LIN {X 0,Y 412.608,Z 386.941,A -85,B 0,C 180,E1 -10561.189,E2 -10561.189} C_VEL
LIN {X 0,Y 413.421,Z 375.355,A -85,B 0,C 180,E1 -10564.715,E2 -10564.715} C_VEL
LIN {X 0,Y 413.845,Z 369.744,A -85,B 0,C 180,E1 -10566.469,E2 -10566.469} C_VEL
LIN {X 0,Y 413.178,Z 364.821,A -85,B 0,C 180,E1 -10568.11,E2 -10568.11} C_VEL
LIN {X 0,Y 411.531,Z 355.758,A -85,B 0,C 180,E1 -10571.286,E2 -10571.286} C_VEL
LIN {X 0,Y 411.225,Z 354.264,A -85,B 0,C 180,E1 -10571.883,E2 -10571.883} C_VEL
LIN {X 0,Y 411.182,Z 354.268,A -85,B 0,C 180,E1 -10575.51,E2 -10575.51} C_VEL
LIN {X 0,Y 411.168,Z 354.271,A -85,B 0,C 180,E1 -10578.772,E2 -10578.772} C_VEL
LIN {X 0,Y 411.21,Z 354.262,A -85,B 0,C 180,E1 -10581.832,E2 -10581.832} C_VEL
LIN {X 0,Y 411.215,Z 354.264,A -85,B 0,C 180,E1 -10585.122,E2 -10585.122} C_VEL
LIN {X 0,Y 411.171,Z 354.266,A -85,B 0,C 180,E1 -10588.003,E2 -10588.003} C_VEL
LIN {X 0,Y 411.223,Z 354.261,A -85,B 0,C 180,E1 -10591.41,E2 -10591.41} C_VEL
LIN {X 0,Y 411.243,Z 354.257,A -85,B 0,C 180,E1 -10593.62,E2 -10593.62} C_VEL
LIN {X 0,Y 411.209,Z 354.265,A -85,B 0,C 180,E1 -10596.853,E2 -10596.853} C_VEL
LIN {X 0,Y 411.22,Z 354.262,A -85,B 0,C 180,E1 -10600.051,E2 -10600.051} C_VEL
LIN {X 0,Y 411.268,Z 354.255,A -85,B 0,C 180,E1 -10603.132,E2 -10603.132} C_VEL
LIN {X 0,Y 411.311,Z 354.252,A -85,B 0,C 180,E1 -10606.896,E2 -10606.896} C_VEL
LIN {X 0,Y 411.298,Z 354.254,A -85,B 0,C 180,E1 -10610.162,E2 -10610.162} C_VEL
LIN {X 0,Y 411.488,Z 354.23,A -85,B 0,C 180,E1 -10612.147,E2 -10612.147} C_VEL
LIN {X 0,Y 411.481,Z 354.231,A -85,B 0,C 180,E1 -10614.118,E2 -10614.118} C_VEL
LIN {X 0,Y 411.517,Z 354.227,A -85,B 0,C 180,E1 -10618.043,E2 -10618.043} C_VEL
LIN {X 0,Y 411.648,Z 354.21,A -85,B 0,C 180,E1 -10620,E2 -10620} C_VEL
LIN {X 0,Y 411.463,Z 354.23,A -85,B 0,C 180,E1 -10622.937,E2 -10622.937} C_VEL
LIN {X 0,Y 411.467,Z 354.229,A -85,B 0,C 180,E1 -10626.867,E2 -10626.867} C_VEL
LIN {X 0,Y 411.3,Z 354.254,A -85,B 0,C 180,E1 -10629.839,E2 -10629.839} C_VEL
LIN {X 0,Y 411.312,Z 354.249,A -85,B 0,C 180,E1 -10633.104,E2 -10633.104} C_VEL
LIN {X 0,Y 411.264,Z 354.255,A -85,B 0,C 180,E1 -10636.889,E2 -10636.889} C_VEL
LIN {X 0,Y 411.237,Z 354.262,A -85,B 0,C 180,E1 -10639.987,E2 -10639.987} C_VEL
LIN {X 0,Y 411.21,Z 354.262,A -85,B 0,C 180,E1 -10643.148,E2 -10643.148} C_VEL
LIN {X 0,Y 411.244,Z 354.258,A -85,B 0,C 180,E1 -10646.381,E2 -10646.381} C_VEL
LIN {X 0,Y 411.207,Z 354.266,A -85,B 0,C 180,E1 -10649.713,E2 -10649.713} C_VEL
LIN {X 0,Y 411.213,Z 354.264,A -85,B 0,C 180,E1 -10653.156,E2 -10653.156} C_VEL
LIN {X 0,Y 411.199,Z 354.263,A -85,B 0,C 180,E1 -10656.553,E2 -10656.553} C_VEL
LIN {X 0,Y 411.221,Z 354.264,A -85,B 0,C 180,E1 -10659.728,E2 -10659.728} C_VEL
LIN {X 0,Y 411.18,Z 354.269,A -85,B 0,C 180,E1 -10663.133,E2 -10663.133} C_VEL
LIN {X 0,Y 411.174,Z 354.267,A -85,B 0,C 180,E1 -10665.881,E2 -10665.881} C_VEL
LIN {X 0,Y 411.17,Z 354.268,A -85,B 0,C 180,E1 -10668.771,E2 -10668.771} C_VEL
LIN {X 0,Y 411.21,Z 354.262,A -85,B 0,C 180,E1 -10671.831,E2 -10671.831} C_VEL
LIN {X 0,Y 411.217,Z 354.265,A -85,B 0,C 180,E1 -10675.121,E2 -10675.121} C_VEL
LIN {X 0,Y 411.172,Z 354.266,A -85,B 0,C 180,E1 -10678.002,E2 -10678.002} C_VEL
LIN {X 0,Y 411.225,Z 354.262,A -85,B 0,C 180,E1 -10681.41,E2 -10681.41} C_VEL
LIN {X 0,Y 411.244,Z 354.258,A -85,B 0,C 180,E1 -10683.619,E2 -10683.619} C_VEL
LIN {X 0,Y 411.21,Z 354.265,A -85,B 0,C 180,E1 -10686.852,E2 -10686.852} C_VEL
LIN {X 0,Y 411.221,Z 354.26,A -85,B 0,C 180,E1 -10690.05,E2 -10690.05} C_VEL
LIN {X 0,Y 411.269,Z 354.257,A -85,B 0,C 180,E1 -10693.131,E2 -10693.131} C_VEL
LIN {X 0,Y 411.312,Z 354.253,A -85,B 0,C 180,E1 -10696.895,E2 -10696.895} C_VEL
LIN {X 0,Y 411.3,Z 354.253,A -85,B 0,C 180,E1 -10700.161,E2 -10700.161} C_VEL
LIN {X 0,Y 411.393,Z 354.352,A -85,B 0,C 180,E1 -10701.301,E2 -10701.301} C_VEL
LIN {X 0,Y 414.802,Z 366.071,A -85,B 0,C 180,E1 -10702.018,E2 -10702.018} C_VEL
LIN {X 0,Y 415.459,Z 369.039,A -85,B 0,C 180,E1 -10702.222,E2 -10702.222} C_VEL
LIN {X 0,Y 414.97,Z 381.177,A -85,B 0,C 180,E1 -10703.069,E2 -10703.069} C_VEL
LIN {X 0,Y 414.349,Z 392.048,A -85,B 0,C 180,E1 -10704.036,E2 -10704.036} C_VEL
LIN {X 0,Y 413.737,Z 401.829,A -85,B 0,C 180,E1 -10705.127,E2 -10705.127} C_VEL
LIN {X 0,Y 413.111,Z 410.706,A -85,B 0,C 180,E1 -10706.342,E2 -10706.342} C_VEL
LIN {X 0,Y 412.467,Z 419.368,A -85,B 0,C 180,E1 -10707.802,E2 -10707.802} C_VEL
LIN {X 0,Y 411.878,Z 426.341,A -85,B 0,C 180,E1 -10709.266,E2 -10709.266} C_VEL
LIN {X 0,Y 411.557,Z 431.041,A -85,B 0,C 180,E1 -10710.489,E2 -10710.489} C_VEL
LIN {X 0,Y 411.291,Z 435.602,A -85,B 0,C 180,E1 -10711.958,E2 -10711.958} C_VEL
LIN {X 0,Y 411.045,Z 438.063,A -85,B 0,C 180,E1 -10712.939,E2 -10712.939} C_VEL
LIN {X 0,Y 410.904,Z 440.046,A -85,B 0,C 180,E1 -10713.922,E2 -10713.922} C_VEL
LIN {X 0,Y 410.94,Z 441.605,A -85,B 0,C 180,E1 -10714.905,E2 -10714.905} C_VEL
LIN {X 0,Y 410.84,Z 443.383,A -85,B 0,C 180,E1 -10716.667,E2 -10716.667} C_VEL
LIN {X 0,Y 410.829,Z 443.911,A -85,B 0,C 180,E1 -10717.865,E2 -10717.865} C_VEL
LIN {X 0,Y 410.835,Z 443.521,A -85,B 0,C 180,E1 -10719.849,E2 -10719.849} C_VEL
LIN {X 0,Y 410.913,Z 442.591,A -85,B 0,C 180,E1 -10720.928,E2 -10720.928} C_VEL
LIN {X 0,Y 410.347,Z 441.725,A -85,B 0,C 180,E1 -10721.738,E2 -10721.738} C_VEL
LIN {X 0,Y 407.723,Z 439.991,A -85,B 0,C 180,E1 -10723.059,E2 -10723.059} C_VEL
LIN {X 0,Y 405.184,Z 437.619,A -85,B 0,C 180,E1 -10724.37,E2 -10724.37} C_VEL
LIN {X 0,Y 404.754,Z 435.61,A -85,B 0,C 180,E1 -10725.154,E2 -10725.154} C_VEL
LIN {X 0,Y 405.227,Z 430.899,A -85,B 0,C 180,E1 -10726.628,E2 -10726.628} C_VEL
LIN {X 0,Y 405.873,Z 424.706,A -85,B 0,C 180,E1 -10728.16,E2 -10728.16} C_VEL
LIN {X 0,Y 406.622,Z 416.874,A -85,B 0,C 180,E1 -10729.696,E2 -10729.696} C_VEL
LIN {X 0,Y 407.382,Z 408.814,A -85,B 0,C 180,E1 -10730.975,E2 -10730.975} C_VEL
LIN {X 0,Y 408.129,Z 398.91,A -85,B 0,C 180,E1 -10732.261,E2 -10732.261} C_VEL
LIN {X 0,Y 408.883,Z 389.085,A -85,B 0,C 180,E1 -10733.286,E2 -10733.286} C_VEL
LIN {X 0,Y 409.693,Z 378.177,A -85,B 0,C 180,E1 -10734.187,E2 -10734.187} C_VEL
LIN {X 0,Y 409.807,Z 371.736,A -85,B 0,C 180,E1 -10734.641,E2 -10734.641} C_VEL
LIN {X 0,Y 405.955,Z 360.3,A -85,B 0,C 180,E1 -10735.523,E2 -10735.523} C_VEL
LIN {X 0,Y 404.213,Z 355.137,A -85,B 0,C 180,E1 -10735.867,E2 -10735.867} C_VEL
LIN {X 0,Y 404.178,Z 355.143,A -85,B 0,C 180,E1 -10739.135,E2 -10739.135} C_VEL
LIN {X 0,Y 404.142,Z 355.149,A -85,B 0,C 180,E1 -10742.621,E2 -10742.621} C_VEL
LIN {X 0,Y 404.181,Z 355.143,A -85,B 0,C 180,E1 -10745.189,E2 -10745.189} C_VEL
LIN {X 0,Y 404.156,Z 355.145,A -85,B 0,C 180,E1 -10748.756,E2 -10748.756} C_VEL
LIN {X 0,Y 404.124,Z 355.146,A -85,B 0,C 180,E1 -10751.599,E2 -10751.599} C_VEL
LIN {X 0,Y 404.148,Z 355.144,A -85,B 0,C 180,E1 -10754.522,E2 -10754.522} C_VEL
LIN {X 0,Y 404.17,Z 355.14,A -85,B 0,C 180,E1 -10757.299,E2 -10757.299} C_VEL
LIN {X 0,Y 404.167,Z 355.141,A -85,B 0,C 180,E1 -10759.955,E2 -10759.955} C_VEL
LIN {X 0,Y 404.14,Z 355.145,A -85,B 0,C 180,E1 -10763.123,E2 -10763.123} C_VEL
LIN {X 0,Y 404.143,Z 355.145,A -85,B 0,C 180,E1 -10766.187,E2 -10766.187} C_VEL
LIN {X 0,Y 404.153,Z 355.118,A -85,B 0,C 180,E1 -10769.715,E2 -10769.715} C_VEL
LIN {X 0,Y 404.193,Z 355.135,A -85,B 0,C 180,E1 -10773.122,E2 -10773.122} C_VEL
LIN {X 0,Y 404.175,Z 355.139,A -85,B 0,C 180,E1 -10775.334,E2 -10775.334} C_VEL
LIN {X 0,Y 404.136,Z 355.145,A -85,B 0,C 180,E1 -10778.58,E2 -10778.58} C_VEL
LIN {X 0,Y 404.207,Z 355.13,A -85,B 0,C 180,E1 -10781.761,E2 -10781.761} C_VEL
LIN {X 0,Y 404.205,Z 355.137,A -85,B 0,C 180,E1 -10784.882,E2 -10784.882} C_VEL
LIN {X 0,Y 404.268,Z 355.129,A -85,B 0,C 180,E1 -10787.959,E2 -10787.959} C_VEL
LIN {X 0,Y 404.43,Z 355.109,A -85,B 0,C 180,E1 -10792.099,E2 -10792.099} C_VEL
LIN {X 0,Y 404.421,Z 355.102,A -85,B 0,C 180,E1 -10794.015,E2 -10794.015} C_VEL
LIN {X 0,Y 404.48,Z 355.102,A -85,B 0,C 180,E1 -10798.008,E2 -10798.008} C_VEL
LIN {X 0,Y 404.61,Z 355.079,A -85,B 0,C 180,E1 -10800,E2 -10800} C_VEL
LIN {X 0,Y 404.42,Z 355.111,A -85,B 0,C 180,E1 -10802.988,E2 -10802.988} C_VEL
LIN {X 0,Y 404.408,Z 355.111,A -85,B 0,C 180,E1 -10806.987,E2 -10806.987} C_VEL
LIN {X 0,Y 404.255,Z 355.124,A -85,B 0,C 180,E1 -10810.012,E2 -10810.012} C_VEL
LIN {X 0,Y 404.262,Z 355.127,A -85,B 0,C 180,E1 -10813.211,E2 -10813.211} C_VEL
LIN {X 0,Y 404.211,Z 355.135,A -85,B 0,C 180,E1 -10817.007,E2 -10817.007} C_VEL
LIN {X 0,Y 404.16,Z 355.141,A -85,B 0,C 180,E1 -10820.352,E2 -10820.352} C_VEL
LIN {X 0,Y 404.166,Z 355.14,A -85,B 0,C 180,E1 -10823.575,E2 -10823.575} C_VEL
LIN {X 0,Y 404.18,Z 355.142,A -85,B 0,C 180,E1 -10825.767,E2 -10825.767} C_VEL
LIN {X 0,Y 404.194,Z 355.142,A -85,B 0,C 180,E1 -10828,E2 -10828} C_VEL
LIN {X 0,Y 404.14,Z 355.147,A -85,B 0,C 180,E1 -10831.559,E2 -10831.559} C_VEL
LIN {X 0,Y 404.182,Z 355.141,A -85,B 0,C 180,E1 -10835.016,E2 -10835.016} C_VEL
LIN {X 0,Y 404.161,Z 355.134,A -85,B 0,C 180,E1 -10838.756,E2 -10838.756} C_VEL
LIN {X 0,Y 404.188,Z 355.131,A -85,B 0,C 180,E1 -10841.611,E2 -10841.611} C_VEL
LIN {X 0,Y 404.196,Z 355.133,A -85,B 0,C 180,E1 -10844.53,E2 -10844.53} C_VEL
LIN {X 0,Y 404.204,Z 355.236,A -85,B 0,C 180,E1 -10846.112,E2 -10846.112} C_VEL
LIN {X 0,Y 405.964,Z 363.942,A -85,B 0,C 180,E1 -10849.616,E2 -10849.616} C_VEL
LIN {X 0,Y 407.483,Z 372.651,A -85,B 0,C 180,E1 -10852.869,E2 -10852.869} C_VEL
LIN {X 0,Y 407.297,Z 376.542,A -85,B 0,C 180,E1 -10854.193,E2 -10854.193} C_VEL
LIN {X 0,Y 406.171,Z 388.134,A -85,B 0,C 180,E1 -10857.979,E2 -10857.979} C_VEL
LIN {X 0,Y 405.429,Z 397.585,A -85,B 0,C 180,E1 -10860.964,E2 -10860.964} C_VEL
LIN {X 0,Y 404.756,Z 408.327,A -85,B 0,C 180,E1 -10864.274,E2 -10864.274} C_VEL
LIN {X 0,Y 404.112,Z 420.824,A -85,B 0,C 180,E1 -10868.044,E2 -10868.044} C_VEL
LIN {X 0,Y 403.632,Z 433.192,A -85,B 0,C 180,E1 -10871.703,E2 -10871.703} C_VEL
LIN {X 0,Y 405.744,Z 447.481,A -85,B 0,C 180,E1 -10872.223,E2 -10872.223} C_VEL
LIN {X 0,Y 406.862,Z 460.005,A -85,B 0,C 180,E1 -10872.843,E2 -10872.843} C_VEL
LIN {X 0,Y 407.384,Z 471.723,A -85,B 0,C 180,E1 -10873.592,E2 -10873.592} C_VEL
LIN {X 0,Y 406.784,Z 481.584,A -85,B 0,C 180,E1 -10874.339,E2 -10874.339} C_VEL
LIN {X 0,Y 405.845,Z 492.192,A -85,B 0,C 180,E1 -10875.33,E2 -10875.33} C_VEL
LIN {X 0,Y 405.155,Z 501.778,A -85,B 0,C 180,E1 -10876.435,E2 -10876.435} C_VEL
LIN {X 0,Y 404.349,Z 510.869,A -85,B 0,C 180,E1 -10877.707,E2 -10877.707} C_VEL
LIN {X 0,Y 403.745,Z 519.623,A -85,B 0,C 180,E1 -10879.216,E2 -10879.216} C_VEL
LIN {X 0,Y 403.409,Z 526.669,A -85,B 0,C 180,E1 -10880.727,E2 -10880.727} C_VEL
LIN {X 0,Y 403.217,Z 533.185,A -85,B 0,C 180,E1 -10882.489,E2 -10882.489} C_VEL
LIN {X 0,Y 403.256,Z 537.494,A -85,B 0,C 180,E1 -10883.998,E2 -10883.998} C_VEL
LIN {X 0,Y 403.23,Z 539.778,A -85,B 0,C 180,E1 -10885.001,E2 -10885.001} C_VEL
LIN {X 0,Y 403.368,Z 541.589,A -85,B 0,C 180,E1 -10886.004,E2 -10886.004} C_VEL
LIN {X 0,Y 403.421,Z 542.973,A -85,B 0,C 180,E1 -10887.005,E2 -10887.005} C_VEL
LIN {X 0,Y 403.367,Z 543.94,A -85,B 0,C 180,E1 -10888.004,E2 -10888.004} C_VEL
LIN {X 0,Y 403.382,Z 544.505,A -85,B 0,C 180,E1 -10889.002,E2 -10889.002} C_VEL
LIN {X 0,Y 403.425,Z 544.63,A -85,B 0,C 180,E1 -10890.001,E2 -10890.001} C_VEL
LIN {X 0,Y 403.401,Z 544.347,A -85,B 0,C 180,E1 -10890.999,E2 -10890.999} C_VEL
LIN {X 0,Y 403.396,Z 543.667,A -85,B 0,C 180,E1 -10891.998,E2 -10891.998} C_VEL
LIN {X 0,Y 403.436,Z 542.583,A -85,B 0,C 180,E1 -10892.996,E2 -10892.996} C_VEL
LIN {X 0,Y 403.373,Z 540.096,A -85,B 0,C 180,E1 -10894.498,E2 -10894.498} C_VEL
LIN {X 0,Y 403.335,Z 536.574,A -85,B 0,C 180,E1 -10896.002,E2 -10896.002} C_VEL
LIN {X 0,Y 403.298,Z 531.93,A -85,B 0,C 180,E1 -10897.511,E2 -10897.511} C_VEL
LIN {X 0,Y 403.419,Z 524.895,A -85,B 0,C 180,E1 -10899.274,E2 -10899.274} C_VEL
LIN {X 0,Y 403.749,Z 517.279,A -85,B 0,C 180,E1 -10900.786,E2 -10900.786} C_VEL
LIN {X 0,Y 404.174,Z 509.526,A -85,B 0,C 180,E1 -10902.045,E2 -10902.045} C_VEL
LIN {X 0,Y 404.837,Z 500.671,A -85,B 0,C 180,E1 -10903.235,E2 -10903.235} C_VEL
LIN {X 0,Y 405.49,Z 491.048,A -85,B 0,C 180,E1 -10904.3,E2 -10904.3} C_VEL
LIN {X 0,Y 406.195,Z 479.805,A -85,B 0,C 180,E1 -10905.3,E2 -10905.3} C_VEL
LIN {X 0,Y 406.698,Z 471.23,A -85,B 0,C 180,E1 -10905.923,E2 -10905.923} C_VEL
LIN {X 0,Y 405.833,Z 458.178,A -85,B 0,C 180,E1 -10906.7,E2 -10906.7} C_VEL
LIN {X 0,Y 404.603,Z 444.289,A -85,B 0,C 180,E1 -10907.307,E2 -10907.307} C_VEL
LIN {X 0,Y 403.522,Z 433.81,A -85,B 0,C 180,E1 -10907.635,E2 -10907.635} C_VEL
LIN {X 0,Y 403.858,Z 422.573,A -85,B 0,C 180,E1 -10910.901,E2 -10910.901} C_VEL
LIN {X 0,Y 404.304,Z 411.609,A -85,B 0,C 180,E1 -10914.111,E2 -10914.111} C_VEL
LIN {X 0,Y 404.952,Z 398.697,A -85,B 0,C 180,E1 -10917.944,E2 -10917.944} C_VEL
LIN {X 0,Y 405.507,Z 389.422,A -85,B 0,C 180,E1 -10920.75,E2 -10920.75} C_VEL
LIN {X 0,Y 406.275,Z 378.033,A -85,B 0,C 180,E1 -10924.27,E2 -10924.27} C_VEL
LIN {X 0,Y 406.852,Z 370.76,A -85,B 0,C 180,E1 -10926.582,E2 -10926.582} C_VEL
LIN {X 0,Y 406.027,Z 365,A -85,B 0,C 180,E1 -10928.546,E2 -10928.546} C_VEL
LIN {X 0,Y 404.417,Z 356.379,A -85,B 0,C 180,E1 -10931.646,E2 -10931.646} C_VEL
LIN {X 0,Y 404.184,Z 355.143,A -85,B 0,C 180,E1 -10932.126,E2 -10932.126} C_VEL
LIN {X 0,Y 404.151,Z 355.144,A -85,B 0,C 180,E1 -10935.478,E2 -10935.478} C_VEL
LIN {X 0,Y 404.123,Z 355.147,A -85,B 0,C 180,E1 -10938.635,E2 -10938.635} C_VEL
LIN {X 0,Y 404.159,Z 355.141,A -85,B 0,C 180,E1 -10941.492,E2 -10941.492} C_VEL
LIN {X 0,Y 404.189,Z 355.141,A -85,B 0,C 180,E1 -10944.984,E2 -10944.984} C_VEL
LIN {X 0,Y 404.147,Z 355.144,A -85,B 0,C 180,E1 -10948.554,E2 -10948.554} C_VEL
LIN {X 0,Y 404.2,Z 355.135,A -85,B 0,C 180,E1 -10952.001,E2 -10952.001} C_VEL
LIN {X 0,Y 404.182,Z 355.137,A -85,B 0,C 180,E1 -10955.335,E2 -10955.335} C_VEL
LIN {X 0,Y 404.144,Z 355.146,A -85,B 0,C 180,E1 -10958.581,E2 -10958.581} C_VEL
LIN {X 0,Y 404.214,Z 355.133,A -85,B 0,C 180,E1 -10961.762,E2 -10961.762} C_VEL
LIN {X 0,Y 404.212,Z 355.136,A -85,B 0,C 180,E1 -10964.882,E2 -10964.882} C_VEL
LIN {X 0,Y 404.261,Z 355.129,A -85,B 0,C 180,E1 -10967.959,E2 -10967.959} C_VEL
LIN {X 0,Y 404.439,Z 355.108,A -85,B 0,C 180,E1 -10972.1,E2 -10972.1} C_VEL
LIN {X 0,Y 404.43,Z 355.109,A -85,B 0,C 180,E1 -10974.015,E2 -10974.015} C_VEL
LIN {X 0,Y 404.486,Z 355.103,A -85,B 0,C 180,E1 -10978.009,E2 -10978.009} C_VEL
LIN {X 0,Y 404.618,Z 355.086,A -85,B 0,C 180,E1 -10980,E2 -10980} C_VEL
LIN {X 0,Y 404.421,Z 355.107,A -85,B 0,C 180,E1 -10982.989,E2 -10982.989} C_VEL
LIN {X 0,Y 404.418,Z 355.107,A -85,B 0,C 180,E1 -10986.987,E2 -10986.987} C_VEL
LIN {X 0,Y 404.265,Z 355.131,A -85,B 0,C 180,E1 -10990.012,E2 -10990.012} C_VEL
LIN {X 0,Y 404.273,Z 355.126,A -85,B 0,C 180,E1 -10993.211,E2 -10993.211} C_VEL
LIN {X 0,Y 404.222,Z 355.132,A -85,B 0,C 180,E1 -10997.007,E2 -10997.007} C_VEL
LIN {X 0,Y 404.17,Z 355.14,A -85,B 0,C 180,E1 -11000.352,E2 -11000.352} C_VEL
LIN {X 0,Y 404.176,Z 355.141,A -85,B 0,C 180,E1 -11003.574,E2 -11003.574} C_VEL
LIN {X 0,Y 404.19,Z 355.14,A -85,B 0,C 180,E1 -11005.766,E2 -11005.766} C_VEL
LIN {X 0,Y 404.201,Z 355.137,A -85,B 0,C 180,E1 -11008,E2 -11008} C_VEL
LIN {X 0,Y 404.146,Z 355.146,A -85,B 0,C 180,E1 -11011.558,E2 -11011.558} C_VEL
LIN {X 0,Y 404.191,Z 355.137,A -85,B 0,C 180,E1 -11015.016,E2 -11015.016} C_VEL
LIN {X 0,Y 404.162,Z 355.139,A -85,B 0,C 180,E1 -11018.757,E2 -11018.757} C_VEL
LIN {X 0,Y 404.13,Z 355.147,A -85,B 0,C 180,E1 -11021.6,E2 -11021.6} C_VEL
LIN {X 0,Y 404.152,Z 355.14,A -85,B 0,C 180,E1 -11024.522,E2 -11024.522} C_VEL
LIN {X 0,Y 404.143,Z 355.146,A -85,B 0,C 180,E1 -11027.295,E2 -11027.295} C_VEL
LIN {X 0,Y 404.175,Z 355.138,A -85,B 0,C 180,E1 -11029.955,E2 -11029.955} C_VEL
LIN {X 0,Y 404.142,Z 355.146,A -85,B 0,C 180,E1 -11033.125,E2 -11033.125} C_VEL
LIN {X 0,Y 404.151,Z 355.141,A -85,B 0,C 180,E1 -11036.187,E2 -11036.187} C_VEL
LIN {X 0,Y 404.152,Z 355.141,A -85,B 0,C 180,E1 -11039.715,E2 -11039.715} C_VEL
LIN {X 0,Y 404.202,Z 355.138,A -85,B 0,C 180,E1 -11043.123,E2 -11043.123} C_VEL
LIN {X 0,Y 404.184,Z 355.139,A -85,B 0,C 180,E1 -11045.334,E2 -11045.334} C_VEL
LIN {X 0,Y 404.145,Z 355.144,A -85,B 0,C 180,E1 -11048.58,E2 -11048.58} C_VEL
LIN {X 0,Y 404.217,Z 355.132,A -85,B 0,C 180,E1 -11051.762,E2 -11051.762} C_VEL
LIN {X 0,Y 404.213,Z 355.137,A -85,B 0,C 180,E1 -11054.882,E2 -11054.882} C_VEL
LIN {X 0,Y 404.263,Z 355.127,A -85,B 0,C 180,E1 -11057.958,E2 -11057.958} C_VEL
LIN {X 0,Y 404.327,Z 355.29,A -85,B 0,C 180,E1 -11061.045,E2 -11061.045} C_VEL
LIN {X 0,Y 407.909,Z 367.47,A -85,B 0,C 180,E1 -11061.811,E2 -11061.811} C_VEL
LIN {X 0,Y 408.548,Z 369.86,A -85,B 0,C 180,E1 -11061.984,E2 -11061.984} C_VEL
LIN {X 0,Y 408.117,Z 381.748,A -85,B 0,C 180,E1 -11062.827,E2 -11062.827} C_VEL
LIN {X 0,Y 407.479,Z 392.676,A -85,B 0,C 180,E1 -11063.811,E2 -11063.811} C_VEL
LIN {X 0,Y 406.897,Z 401.527,A -85,B 0,C 180,E1 -11064.797,E2 -11064.797} C_VEL
LIN {X 0,Y 406.268,Z 410.621,A -85,B 0,C 180,E1 -11066.031,E2 -11066.031} C_VEL
LIN {X 0,Y 405.564,Z 419.448,A -85,B 0,C 180,E1 -11067.516,E2 -11067.516} C_VEL
LIN {X 0,Y 404.945,Z 426.573,A -85,B 0,C 180,E1 -11069.005,E2 -11069.005} C_VEL
LIN {X 0,Y 404.531,Z 432.269,A -85,B 0,C 180,E1 -11070.497,E2 -11070.497} C_VEL
LIN {X 0,Y 404.242,Z 436.756,A -85,B 0,C 180,E1 -11071.992,E2 -11071.992} C_VEL
LIN {X 0,Y 403.989,Z 439.148,A -85,B 0,C 180,E1 -11072.991,E2 -11072.991} C_VEL
LIN {X 0,Y 403.863,Z 441.096,A -85,B 0,C 180,E1 -11073.991,E2 -11073.991} C_VEL
LIN {X 0,Y 403.896,Z 442.623,A -85,B 0,C 180,E1 -11074.99,E2 -11074.99} C_VEL
LIN {X 0,Y 403.839,Z 443.752,A -85,B 0,C 180,E1 -11075.993,E2 -11075.993} C_VEL
LIN {X 0,Y 403.781,Z 444.803,A -85,B 0,C 180,E1 -11078.003,E2 -11078.003} C_VEL
LIN {X 0,Y 403.772,Z 444.769,A -85,B 0,C 180,E1 -11079.012,E2 -11079.012} C_VEL
LIN {X 0,Y 403.823,Z 444.322,A -85,B 0,C 180,E1 -11080.022,E2 -11080.022} C_VEL
LIN {X 0,Y 404.073,Z 442.198,A -85,B 0,C 180,E1 -11082.046,E2 -11082.046} C_VEL
LIN {X 0,Y 404.297,Z 440.208,A -85,B 0,C 180,E1 -11083.227,E2 -11083.227} C_VEL
LIN {X 0,Y 404.736,Z 435.778,A -85,B 0,C 180,E1 -11085.097,E2 -11085.097} C_VEL
LIN {X 0,Y 404.754,Z 435.61,A -85,B 0,C 180,E1 -11085.154,E2 -11085.154} C_VEL
LIN {X 0,Y 404.339,Z 433.425,A -85,B 0,C 180,E1 -11085.929,E2 -11085.929} C_VEL
LIN {X 0,Y 401.929,Z 429.615,A -85,B 0,C 180,E1 -11087.19,E2 -11087.19} C_VEL
LIN {X 0,Y 399.613,Z 425.244,A -85,B 0,C 180,E1 -11088.419,E2 -11088.419} C_VEL
LIN {X 0,Y 399.34,Z 422.036,A -85,B 0,C 180,E1 -11089.129,E2 -11089.129} C_VEL
LIN {X 0,Y 400.197,Z 414.087,A -85,B 0,C 180,E1 -11090.562,E2 -11090.562} C_VEL
LIN {X 0,Y 400.992,Z 405.578,A -85,B 0,C 180,E1 -11091.814,E2 -11091.814} C_VEL
LIN {X 0,Y 401.74,Z 396.558,A -85,B 0,C 180,E1 -11092.906,E2 -11092.906} C_VEL
LIN {X 0,Y 402.48,Z 386.284,A -85,B 0,C 180,E1 -11093.921,E2 -11093.921} C_VEL
LIN {X 0,Y 403.209,Z 374.639,A -85,B 0,C 180,E1 -11094.826,E2 -11094.826} C_VEL
LIN {X 0,Y 401.693,Z 369.084,A -85,B 0,C 180,E1 -11095.284,E2 -11095.284} C_VEL
LIN {X 0,Y 397.208,Z 356.375,A -85,B 0,C 180,E1 -11096.219,E2 -11096.219} C_VEL
LIN {X 0,Y 397.153,Z 356.017,A -85,B 0,C 180,E1 -11096.256,E2 -11096.256} C_VEL
LIN {X 0,Y 397.123,Z 356.019,A -85,B 0,C 180,E1 -11098.543,E2 -11098.543} C_VEL
LIN {X 0,Y 397.08,Z 356.029,A -85,B 0,C 180,E1 -11102.071,E2 -11102.071} C_VEL
LIN {X 0,Y 397.12,Z 356.023,A -85,B 0,C 180,E1 -11105.502,E2 -11105.502} C_VEL
LIN {X 0,Y 397.131,Z 356.019,A -85,B 0,C 180,E1 -11108.861,E2 -11108.861} C_VEL
LIN {X 0,Y 397.071,Z 356.024,A -85,B 0,C 180,E1 -11112.266,E2 -11112.266} C_VEL
LIN {X 0,Y 397.088,Z 356.024,A -85,B 0,C 180,E1 -11115.068,E2 -11115.068} C_VEL
LIN {X 0,Y 397.109,Z 356.022,A -85,B 0,C 180,E1 -11118.013,E2 -11118.013} C_VEL
LIN {X 0,Y 397.137,Z 356.018,A -85,B 0,C 180,E1 -11121.136,E2 -11121.136} C_VEL
LIN {X 0,Y 397.119,Z 356.019,A -85,B 0,C 180,E1 -11124.496,E2 -11124.496} C_VEL
LIN {X 0,Y 397.109,Z 356.012,A -85,B 0,C 180,E1 -11127.931,E2 -11127.931} C_VEL
LIN {X 0,Y 397.125,Z 356.004,A -85,B 0,C 180,E1 -11131.456,E2 -11131.456} C_VEL
LIN {X 0,Y 397.15,Z 356.016,A -85,B 0,C 180,E1 -11134.487,E2 -11134.487} C_VEL
LIN {X 0,Y 397.106,Z 356.013,A -85,B 0,C 180,E1 -11137.085,E2 -11137.085} C_VEL
LIN {X 0,Y 397.145,Z 356.016,A -85,B 0,C 180,E1 -11140.352,E2 -11140.352} C_VEL
LIN {X 0,Y 397.163,Z 356.012,A -85,B 0,C 180,E1 -11143.553,E2 -11143.553} C_VEL
LIN {X 0,Y 397.225,Z 356.004,A -85,B 0,C 180,E1 -11146.702,E2 -11146.702} C_VEL
LIN {X 0,Y 397.227,Z 356.003,A -85,B 0,C 180,E1 -11149.809,E2 -11149.809} C_VEL
LIN {X 0,Y 397.36,Z 355.987,A -85,B 0,C 180,E1 -11152.888,E2 -11152.888} C_VEL
LIN {X 0,Y 397.253,Z 355.996,A -85,B 0,C 180,E1 -11154.925,E2 -11154.925} C_VEL
LIN {X 0,Y 397.449,Z 355.978,A -85,B 0,C 180,E1 -11157.973,E2 -11157.973} C_VEL
LIN {X 0,Y 397.579,Z 355.954,A -85,B 0,C 180,E1 -11160,E2 -11160} C_VEL
LIN {X 0,Y 397.379,Z 355.988,A -85,B 0,C 180,E1 -11163.041,E2 -11163.041} C_VEL
LIN {X 0,Y 397.36,Z 355.99,A -85,B 0,C 180,E1 -11167.112,E2 -11167.112} C_VEL
LIN {X 0,Y 397.214,Z 356.002,A -85,B 0,C 180,E1 -11170.191,E2 -11170.191} C_VEL
LIN {X 0,Y 397.222,Z 356.003,A -85,B 0,C 180,E1 -11173.321,E2 -11173.321} C_VEL
LIN {X 0,Y 397.177,Z 356.01,A -85,B 0,C 180,E1 -11177.155,E2 -11177.155} C_VEL
LIN {X 0,Y 397.098,Z 356.019,A -85,B 0,C 180,E1 -11180.73,E2 -11180.73} C_VEL
LIN {X 0,Y 397.129,Z 356.017,A -85,B 0,C 180,E1 -11184.018,E2 -11184.018} C_VEL
LIN {X 0,Y 397.191,Z 356.014,A -85,B 0,C 180,E1 -11187.39,E2 -11187.39} C_VEL
LIN {X 0,Y 397.081,Z 356.026,A -85,B 0,C 180,E1 -11190.882,E2 -11190.882} C_VEL
LIN {X 0,Y 397.123,Z 356.02,A -85,B 0,C 180,E1 -11194.494,E2 -11194.494} C_VEL
LIN {X 0,Y 397.107,Z 356.012,A -85,B 0,C 180,E1 -11198.274,E2 -11198.274} C_VEL
LIN {X 0,Y 397.153,Z 356.008,A -85,B 0,C 180,E1 -11201.994,E2 -11201.994} C_VEL
LIN {X 0,Y 397.16,Z 356.015,A -85,B 0,C 180,E1 -11205.58,E2 -11205.58} C_VEL
LIN {X 0,Y 398.544,Z 362.992,A -85,B 0,C 180,E1 -11208.542,E2 -11208.542} C_VEL
LIN {X 0,Y 399.907,Z 370.296,A -85,B 0,C 180,E1 -11211.401,E2 -11211.401} C_VEL
LIN {X 0,Y 400.549,Z 374.033,A -85,B 0,C 180,E1 -11212.797,E2 -11212.797} C_VEL
LIN {X 0,Y 400.301,Z 378.101,A -85,B 0,C 180,E1 -11214.21,E2 -11214.21} C_VEL
LIN {X 0,Y 399.114,Z 389.845,A -85,B 0,C 180,E1 -11218.112,E2 -11218.112} C_VEL
LIN {X 0,Y 398.228,Z 400.526,A -85,B 0,C 180,E1 -11221.544,E2 -11221.544} C_VEL
LIN {X 0,Y 397.545,Z 411.22,A -85,B 0,C 180,E1 -11224.896,E2 -11224.896} C_VEL
LIN {X 0,Y 396.997,Z 421.885,A -85,B 0,C 180,E1 -11228.177,E2 -11228.177} C_VEL
LIN {X 0,Y 396.586,Z 432.153,A -85,B 0,C 180,E1 -11231.299,E2 -11231.299} C_VEL
LIN {X 0,Y 398.879,Z 447.676,A -85,B 0,C 180,E1 -11231.902,E2 -11231.902} C_VEL
LIN {X 0,Y 400.004,Z 460.144,A -85,B 0,C 180,E1 -11232.556,E2 -11232.556} C_VEL
LIN {X 0,Y 400.505,Z 473.18,A -85,B 0,C 180,E1 -11233.433,E2 -11233.433} C_VEL
LIN {X 0,Y 399.64,Z 484.018,A -85,B 0,C 180,E1 -11234.314,E2 -11234.314} C_VEL
LIN {X 0,Y 398.661,Z 495.139,A -85,B 0,C 180,E1 -11235.451,E2 -11235.451} C_VEL
LIN {X 0,Y 397.947,Z 505.123,A -85,B 0,C 180,E1 -11236.728,E2 -11236.728} C_VEL
LIN {X 0,Y 397.167,Z 513.331,A -85,B 0,C 180,E1 -11238,E2 -11238} C_VEL
LIN {X 0,Y 396.549,Z 521.439,A -85,B 0,C 180,E1 -11239.534,E2 -11239.534} C_VEL
LIN {X 0,Y 396.31,Z 526.97,A -85,B 0,C 180,E1 -11240.817,E2 -11240.817} C_VEL
LIN {X 0,Y 396.162,Z 532.422,A -85,B 0,C 180,E1 -11242.355,E2 -11242.355} C_VEL
LIN {X 0,Y 396.18,Z 536.702,A -85,B 0,C 180,E1 -11243.891,E2 -11243.891} C_VEL
LIN {X 0,Y 396.16,Z 538.966,A -85,B 0,C 180,E1 -11244.912,E2 -11244.912} C_VEL
LIN {X 0,Y 396.302,Z 540.763,A -85,B 0,C 180,E1 -11245.933,E2 -11245.933} C_VEL
LIN {X 0,Y 396.373,Z 542.138,A -85,B 0,C 180,E1 -11246.952,E2 -11246.952} C_VEL
LIN {X 0,Y 396.314,Z 543.093,A -85,B 0,C 180,E1 -11247.968,E2 -11247.968} C_VEL
LIN {X 0,Y 396.332,Z 543.64,A -85,B 0,C 180,E1 -11248.985,E2 -11248.985} C_VEL
LIN {X 0,Y 396.38,Z 543.752,A -85,B 0,C 180,E1 -11250.001,E2 -11250.001} C_VEL
LIN {X 0,Y 396.354,Z 543.457,A -85,B 0,C 180,E1 -11251.017,E2 -11251.017} C_VEL
LIN {X 0,Y 396.347,Z 542.765,A -85,B 0,C 180,E1 -11252.033,E2 -11252.033} C_VEL
LIN {X 0,Y 396.39,Z 541.661,A -85,B 0,C 180,E1 -11253.05,E2 -11253.05} C_VEL
LIN {X 0,Y 396.312,Z 539.152,A -85,B 0,C 180,E1 -11254.578,E2 -11254.578} C_VEL
LIN {X 0,Y 396.276,Z 535.605,A -85,B 0,C 180,E1 -11256.109,E2 -11256.109} C_VEL
LIN {X 0,Y 396.224,Z 530.926,A -85,B 0,C 180,E1 -11257.646,E2 -11257.646} C_VEL
LIN {X 0,Y 396.372,Z 523.845,A -85,B 0,C 180,E1 -11259.44,E2 -11259.44} C_VEL
LIN {X 0,Y 396.733,Z 516.19,A -85,B 0,C 180,E1 -11260.979,E2 -11260.979} C_VEL
LIN {X 0,Y 397.173,Z 508.392,A -85,B 0,C 180,E1 -11262.26,E2 -11262.26} C_VEL
LIN {X 0,Y 397.794,Z 499.095,A -85,B 0,C 180,E1 -11263.521,E2 -11263.521} C_VEL
LIN {X 0,Y 398.633,Z 488.456,A -85,B 0,C 180,E1 -11264.682,E2 -11264.682} C_VEL
LIN {X 0,Y 399.438,Z 476.824,A -85,B 0,C 180,E1 -11265.696,E2 -11265.696} C_VEL
LIN {X 0,Y 399.527,Z 469.666,A -85,B 0,C 180,E1 -11266.216,E2 -11266.216} C_VEL
LIN {X 0,Y 398.821,Z 457.782,A -85,B 0,C 180,E1 -11266.935,E2 -11266.935} C_VEL
LIN {X 0,Y 397.613,Z 444.053,A -85,B 0,C 180,E1 -11267.554,E2 -11267.554} C_VEL
LIN {X 0,Y 396.446,Z 432.949,A -85,B 0,C 180,E1 -11267.907,E2 -11267.907} C_VEL
LIN {X 0,Y 396.825,Z 421.591,A -85,B 0,C 180,E1 -11271.289,E2 -11271.289} C_VEL
LIN {X 0,Y 397.286,Z 410.654,A -85,B 0,C 180,E1 -11274.565,E2 -11274.565} C_VEL
LIN {X 0,Y 398.008,Z 397.772,A -85,B 0,C 180,E1 -11278.475,E2 -11278.475} C_VEL
LIN {X 0,Y 398.701,Z 386.631,A -85,B 0,C 180,E1 -11281.926,E2 -11281.926} C_VEL
LIN {X 0,Y 399.58,Z 375.478,A -85,B 0,C 180,E1 -11285.481,E2 -11285.481} C_VEL
LIN {X 0,Y 399.871,Z 371.759,A -85,B 0,C 180,E1 -11286.697,E2 -11286.697} C_VEL
LIN {X 0,Y 398.782,Z 364.74,A -85,B 0,C 180,E1 -11289.155,E2 -11289.155} C_VEL
LIN {X 0,Y 397.131,Z 356.02,A -85,B 0,C 180,E1 -11292.431,E2 -11292.431} C_VEL
LIN {X 0,Y 397.105,Z 356.023,A -85,B 0,C 180,E1 -11296.352,E2 -11296.352} C_VEL
LIN {X 0,Y 397.105,Z 356.019,A -85,B 0,C 180,E1 -11299.555,E2 -11299.555} C_VEL
LIN {X 0,Y 397.099,Z 356.023,A -85,B 0,C 180,E1 -11302.791,E2 -11302.791} C_VEL
LIN {X 0,Y 397.123,Z 356.017,A -85,B 0,C 180,E1 -11306.283,E2 -11306.283} C_VEL
LIN {X 0,Y 397.11,Z 356.018,A -85,B 0,C 180,E1 -11310.136,E2 -11310.136} C_VEL
LIN {X 0,Y 397.199,Z 356.01,A -85,B 0,C 180,E1 -11312.61,E2 -11312.61} C_VEL
LIN {X 0,Y 397.138,Z 356.014,A -85,B 0,C 180,E1 -11315.982,E2 -11315.982} C_VEL
LIN {X 0,Y 397.144,Z 356.013,A -85,B 0,C 180,E1 -11319.705,E2 -11319.705} C_VEL
LIN {X 0,Y 397.187,Z 356.011,A -85,B 0,C 180,E1 -11322.845,E2 -11322.845} C_VEL
LIN {X 0,Y 397.234,Z 356.006,A -85,B 0,C 180,E1 -11326.703,E2 -11326.703} C_VEL
LIN {X 0,Y 397.223,Z 356.004,A -85,B 0,C 180,E1 -11329.809,E2 -11329.809} C_VEL
LIN {X 0,Y 397.37,Z 355.987,A -85,B 0,C 180,E1 -11332.888,E2 -11332.888} C_VEL
LIN {X 0,Y 397.259,Z 356,A -85,B 0,C 180,E1 -11334.925,E2 -11334.925} C_VEL
LIN {X 0,Y 397.455,Z 355.978,A -85,B 0,C 180,E1 -11337.974,E2 -11337.974} C_VEL
LIN {X 0,Y 397.587,Z 355.962,A -85,B 0,C 180,E1 -11340,E2 -11340} C_VEL
LIN {X 0,Y 397.381,Z 355.984,A -85,B 0,C 180,E1 -11343.042,E2 -11343.042} C_VEL
LIN {X 0,Y 397.37,Z 355.985,A -85,B 0,C 180,E1 -11347.112,E2 -11347.112} C_VEL
LIN {X 0,Y 397.224,Z 356.007,A -85,B 0,C 180,E1 -11350.191,E2 -11350.191} C_VEL
LIN {X 0,Y 397.233,Z 356.003,A -85,B 0,C 180,E1 -11353.321,E2 -11353.321} C_VEL
LIN {X 0,Y 397.188,Z 356.008,A -85,B 0,C 180,E1 -11357.155,E2 -11357.155} C_VEL
LIN {X 0,Y 397.109,Z 356.017,A -85,B 0,C 180,E1 -11360.73,E2 -11360.73} C_VEL
LIN {X 0,Y 397.139,Z 356.018,A -85,B 0,C 180,E1 -11364.018,E2 -11364.018} C_VEL
LIN {X 0,Y 397.201,Z 356.01,A -85,B 0,C 180,E1 -11367.39,E2 -11367.39} C_VEL
LIN {X 0,Y 397.085,Z 356.021,A -85,B 0,C 180,E1 -11370.882,E2 -11370.882} C_VEL
LIN {X 0,Y 397.132,Z 356.015,A -85,B 0,C 180,E1 -11374.493,E2 -11374.493} C_VEL
LIN {X 0,Y 397.11,Z 356.017,A -85,B 0,C 180,E1 -11378.275,E2 -11378.275} C_VEL
LIN {X 0,Y 397.095,Z 356.021,A -85,B 0,C 180,E1 -11380.909,E2 -11380.909} C_VEL
LIN {X 0,Y 397.107,Z 356.021,A -85,B 0,C 180,E1 -11383.648,E2 -11383.648} C_VEL
LIN {X 0,Y 397.108,Z 356.018,A -85,B 0,C 180,E1 -11386.521,E2 -11386.521} C_VEL
LIN {X 0,Y 397.12,Z 356.016,A -85,B 0,C 180,E1 -11390.423,E2 -11390.423} C_VEL
LIN {X 0,Y 397.114,Z 356.017,A -85,B 0,C 180,E1 -11394.265,E2 -11394.265} C_VEL
LIN {X 0,Y 397.121,Z 356.019,A -85,B 0,C 180,E1 -11396.727,E2 -11396.727} C_VEL
LIN {X 0,Y 397.131,Z 356.015,A -85,B 0,C 180,E1 -11400.296,E2 -11400.296} C_VEL
LIN {X 0,Y 397.201,Z 356.008,A -85,B 0,C 180,E1 -11402.61,E2 -11402.61} C_VEL
LIN {X 0,Y 397.139,Z 356.014,A -85,B 0,C 180,E1 -11405.981,E2 -11405.981} C_VEL
LIN {X 0,Y 397.145,Z 356.013,A -85,B 0,C 180,E1 -11409.704,E2 -11409.704} C_VEL
LIN {X 0,Y 397.188,Z 356.012,A -85,B 0,C 180,E1 -11412.844,E2 -11412.844} C_VEL
LIN {X 0,Y 397.235,Z 356.006,A -85,B 0,C 180,E1 -11416.702,E2 -11416.702} C_VEL
LIN {X 0,Y 397.242,Z 356.005,A -85,B 0,C 180,E1 -11420.58,E2 -11420.58} C_VEL
LIN {X 0,Y 397.24,Z 356.062,A -85,B 0,C 180,E1 -11420.773,E2 -11420.773} C_VEL
LIN {X 0,Y 400.849,Z 368.071,A -85,B 0,C 180,E1 -11421.544,E2 -11421.544} C_VEL
LIN {X 0,Y 401.736,Z 371.82,A -85,B 0,C 180,E1 -11421.819,E2 -11421.819} C_VEL
LIN {X 0,Y 401.18,Z 383.855,A -85,B 0,C 180,E1 -11422.703,E2 -11422.703} C_VEL
LIN {X 0,Y 400.502,Z 394.506,A -85,B 0,C 180,E1 -11423.703,E2 -11423.703} C_VEL
LIN {X 0,Y 399.807,Z 405.099,A -85,B 0,C 180,E1 -11424.957,E2 -11424.957} C_VEL
LIN {X 0,Y 399.154,Z 413.721,A -85,B 0,C 180,E1 -11426.213,E2 -11426.213} C_VEL
LIN {X 0,Y 398.458,Z 422.136,A -85,B 0,C 180,E1 -11427.725,E2 -11427.725} C_VEL
LIN {X 0,Y 397.91,Z 427.88,A -85,B 0,C 180,E1 -11428.987,E2 -11428.987} C_VEL
LIN {X 0,Y 397.504,Z 433.472,A -85,B 0,C 180,E1 -11430.506,E2 -11430.506} C_VEL
LIN {X 0,Y 397.194,Z 437.884,A -85,B 0,C 180,E1 -11432.027,E2 -11432.027} C_VEL
LIN {X 0,Y 396.935,Z 440.23,A -85,B 0,C 180,E1 -11433.044,E2 -11433.044} C_VEL
LIN {X 0,Y 396.821,Z 442.143,A -85,B 0,C 180,E1 -11434.062,E2 -11434.062} C_VEL
LIN {X 0,Y 396.853,Z 443.635,A -85,B 0,C 180,E1 -11435.079,E2 -11435.079} C_VEL
LIN {X 0,Y 396.762,Z 445.385,A -85,B 0,C 180,E1 -11437.122,E2 -11437.122} C_VEL
LIN {X 0,Y 396.746,Z 445.623,A -85,B 0,C 180,E1 -11439.173,E2 -11439.173} C_VEL
LIN {X 0,Y 396.882,Z 444.225,A -85,B 0,C 180,E1 -11441.232,E2 -11441.232} C_VEL
LIN {X 0,Y 397.103,Z 442.929,A -85,B 0,C 180,E1 -11442.261,E2 -11442.261} C_VEL
LIN {X 0,Y 397.397,Z 440.173,A -85,B 0,C 180,E1 -11443.811,E2 -11443.811} C_VEL
LIN {X 0,Y 397.82,Z 436.373,A -85,B 0,C 180,E1 -11445.366,E2 -11445.366} C_VEL
LIN {X 0,Y 398.36,Z 431.416,A -85,B 0,C 180,E1 -11446.923,E2 -11446.923} C_VEL
LIN {X 0,Y 399.037,Z 425.118,A -85,B 0,C 180,E1 -11448.482,E2 -11448.482} C_VEL
LIN {X 0,Y 399.34,Z 422.036,A -85,B 0,C 180,E1 -11449.129,E2 -11449.129} C_VEL
LIN {X 0,Y 399.092,Z 418.635,A -85,B 0,C 180,E1 -11449.821,E2 -11449.821} C_VEL
LIN {X 0,Y 396.925,Z 412.956,A -85,B 0,C 180,E1 -11450.955,E2 -11450.955} C_VEL
LIN {X 0,Y 394.787,Z 406.748,A -85,B 0,C 180,E1 -11452.03,E2 -11452.03} C_VEL
LIN {X 0,Y 394.569,Z 402.473,A -85,B 0,C 180,E1 -11452.619,E2 -11452.619} C_VEL
LIN {X 0,Y 395.463,Z 391.404,A -85,B 0,C 180,E1 -11453.847,E2 -11453.847} C_VEL
LIN {X 0,Y 396.388,Z 379.988,A -85,B 0,C 180,E1 -11454.829,E2 -11454.829} C_VEL
LIN {X 0,Y 396.446,Z 375.37,A -85,B 0,C 180,E1 -11455.179,E2 -11455.179} C_VEL
LIN {X 0,Y 392.58,Z 363.949,A -85,B 0,C 180,E1 -11456.133,E2 -11456.133} C_VEL
LIN {X 0,Y 390.117,Z 356.894,A -85,B 0,C 180,E1 -11456.662,E2 -11456.662} C_VEL
LIN {X 0,Y 390.048,Z 356.905,A -85,B 0,C 180,E1 -11460.13,E2 -11460.13} C_VEL
LIN {X 0,Y 390.069,Z 356.896,A -85,B 0,C 180,E1 -11464.024,E2 -11464.024} C_VEL
LIN {X 0,Y 390.044,Z 356.902,A -85,B 0,C 180,E1 -11467.55,E2 -11467.55} C_VEL
LIN {X 0,Y 390.056,Z 356.9,A -85,B 0,C 180,E1 -11470.821,E2 -11470.821} C_VEL
LIN {X 0,Y 390.056,Z 356.899,A -85,B 0,C 180,E1 -11473.886,E2 -11473.886} C_VEL
LIN {X 0,Y 390.079,Z 356.897,A -85,B 0,C 180,E1 -11477.619,E2 -11477.619} C_VEL
LIN {X 0,Y 390.094,Z 356.895,A -85,B 0,C 180,E1 -11480.908,E2 -11480.908} C_VEL
LIN {X 0,Y 390.084,Z 356.896,A -85,B 0,C 180,E1 -11484.792,E2 -11484.792} C_VEL
LIN {X 0,Y 390.045,Z 356.886,A -85,B 0,C 180,E1 -11488.497,E2 -11488.497} C_VEL
LIN {X 0,Y 390.114,Z 356.882,A -85,B 0,C 180,E1 -11492.069,E2 -11492.069} C_VEL
LIN {X 0,Y 390.077,Z 356.894,A -85,B 0,C 180,E1 -11495.519,E2 -11495.519} C_VEL
LIN {X 0,Y 390.053,Z 356.899,A -85,B 0,C 180,E1 -11498.877,E2 -11498.877} C_VEL
LIN {X 0,Y 390.125,Z 356.883,A -85,B 0,C 180,E1 -11502.166,E2 -11502.166} C_VEL
LIN {X 0,Y 390.144,Z 356.89,A -85,B 0,C 180,E1 -11505.392,E2 -11505.392} C_VEL
LIN {X 0,Y 390.158,Z 356.887,A -85,B 0,C 180,E1 -11508.571,E2 -11508.571} C_VEL
LIN {X 0,Y 390.34,Z 356.864,A -85,B 0,C 180,E1 -11511.993,E2 -11511.993} C_VEL
LIN {X 0,Y 390.225,Z 356.871,A -85,B 0,C 180,E1 -11514.833,E2 -11514.833} C_VEL
LIN {X 0,Y 390.417,Z 356.854,A -85,B 0,C 180,E1 -11517.937,E2 -11517.937} C_VEL
LIN {X 0,Y 390.549,Z 356.829,A -85,B 0,C 180,E1 -11520,E2 -11520} C_VEL
LIN {X 0,Y 390.313,Z 356.868,A -85,B 0,C 180,E1 -11523.096,E2 -11523.096} C_VEL
LIN {X 0,Y 390.327,Z 356.863,A -85,B 0,C 180,E1 -11526.202,E2 -11526.202} C_VEL
LIN {X 0,Y 390.31,Z 356.867,A -85,B 0,C 180,E1 -11528.282,E2 -11528.282} C_VEL
LIN {X 0,Y 390.167,Z 356.885,A -85,B 0,C 180,E1 -11532.483,E2 -11532.483} C_VEL
LIN {X 0,Y 390.135,Z 356.889,A -85,B 0,C 180,E1 -11535.677,E2 -11535.677} C_VEL
LIN {X 0,Y 390.102,Z 356.894,A -85,B 0,C 180,E1 -11538.922,E2 -11538.922} C_VEL
LIN {X 0,Y 390.036,Z 356.904,A -85,B 0,C 180,E1 -11542.234,E2 -11542.234} C_VEL
LIN {X 0,Y 390.115,Z 356.894,A -85,B 0,C 180,E1 -11545.744,E2 -11545.744} C_VEL
LIN {X 0,Y 390.062,Z 356.902,A -85,B 0,C 180,E1 -11549.109,E2 -11549.109} C_VEL
LIN {X 0,Y 390.04,Z 356.902,A -85,B 0,C 180,E1 -11552.722,E2 -11552.722} C_VEL
LIN {X 0,Y 390.054,Z 356.898,A -85,B 0,C 180,E1 -11555.826,E2 -11555.826} C_VEL
LIN {X 0,Y 390.072,Z 356.891,A -85,B 0,C 180,E1 -11559.22,E2 -11559.22} C_VEL
LIN {X 0,Y 390.119,Z 356.887,A -85,B 0,C 180,E1 -11562.387,E2 -11562.387} C_VEL
LIN {X 0,Y 390.136,Z 357.092,A -85,B 0,C 180,E1 -11565.278,E2 -11565.278} C_VEL
LIN {X 0,Y 391.586,Z 364.386,A -85,B 0,C 180,E1 -11568.391,E2 -11568.391} C_VEL
LIN {X 0,Y 392.938,Z 371.527,A -85,B 0,C 180,E1 -11571.245,E2 -11571.245} C_VEL
LIN {X 0,Y 393.619,Z 376.478,A -85,B 0,C 180,E1 -11573.11,E2 -11573.11} C_VEL
LIN {X 0,Y 392.621,Z 385.711,A -85,B 0,C 180,E1 -11576.297,E2 -11576.297} C_VEL
LIN {X 0,Y 391.64,Z 396.346,A -85,B 0,C 180,E1 -11579.838,E2 -11579.838} C_VEL
LIN {X 0,Y 390.844,Z 407,A -85,B 0,C 180,E1 -11583.287,E2 -11583.287} C_VEL
LIN {X 0,Y 390.088,Z 419.516,A -85,B 0,C 180,E1 -11587.247,E2 -11587.247} C_VEL
LIN {X 0,Y 389.527,Z 431.288,A -85,B 0,C 180,E1 -11590.913,E2 -11590.913} C_VEL
LIN {X 0,Y 391.757,Z 445.409,A -85,B 0,C 180,E1 -11591.461,E2 -11591.461} C_VEL
LIN {X 0,Y 392.971,Z 457.096,A -85,B 0,C 180,E1 -11592.066,E2 -11592.066} C_VEL
LIN {X 0,Y 393.42,Z 469.323,A -85,B 0,C 180,E1 -11592.858,E2 -11592.858} C_VEL
LIN {X 0,Y 393.518,Z 476.174,A -85,B 0,C 180,E1 -11593.397,E2 -11593.397} C_VEL
LIN {X 0,Y 392.412,Z 487.532,A -85,B 0,C 180,E1 -11594.417,E2 -11594.417} C_VEL
LIN {X 0,Y 391.414,Z 498.24,A -85,B 0,C 180,E1 -11595.629,E2 -11595.629} C_VEL
LIN {X 0,Y 390.62,Z 507.966,A -85,B 0,C 180,E1 -11597.004,E2 -11597.004} C_VEL
LIN {X 0,Y 389.818,Z 516.927,A -85,B 0,C 180,E1 -11598.562,E2 -11598.562} C_VEL
LIN {X 0,Y 389.33,Z 524.166,A -85,B 0,C 180,E1 -11600.126,E2 -11600.126} C_VEL
LIN {X 0,Y 389.139,Z 529.994,A -85,B 0,C 180,E1 -11601.693,E2 -11601.693} C_VEL
LIN {X 0,Y 389.075,Z 535.112,A -85,B 0,C 180,E1 -11603.457,E2 -11603.457} C_VEL
LIN {X 0,Y 389.095,Z 538.155,A -85,B 0,C 180,E1 -11604.819,E2 -11604.819} C_VEL
LIN {X 0,Y 389.239,Z 539.94,A -85,B 0,C 180,E1 -11605.859,E2 -11605.859} C_VEL
LIN {X 0,Y 389.325,Z 541.305,A -85,B 0,C 180,E1 -11606.896,E2 -11606.896} C_VEL
LIN {X 0,Y 389.26,Z 542.249,A -85,B 0,C 180,E1 -11607.931,E2 -11607.931} C_VEL
LIN {X 0,Y 389.282,Z 542.772,A -85,B 0,C 180,E1 -11608.966,E2 -11608.966} C_VEL
LIN {X 0,Y 389.334,Z 542.873,A -85,B 0,C 180,E1 -11610.001,E2 -11610.001} C_VEL
LIN {X 0,Y 389.306,Z 542.566,A -85,B 0,C 180,E1 -11611.035,E2 -11611.035} C_VEL
LIN {X 0,Y 389.298,Z 541.862,A -85,B 0,C 180,E1 -11612.07,E2 -11612.07} C_VEL
LIN {X 0,Y 389.344,Z 540.735,A -85,B 0,C 180,E1 -11613.105,E2 -11613.105} C_VEL
LIN {X 0,Y 389.252,Z 538.203,A -85,B 0,C 180,E1 -11614.661,E2 -11614.661} C_VEL
LIN {X 0,Y 389.152,Z 533.444,A -85,B 0,C 180,E1 -11616.641,E2 -11616.641} C_VEL
LIN {X 0,Y 389.206,Z 528.054,A -85,B 0,C 180,E1 -11618.307,E2 -11618.307} C_VEL
LIN {X 0,Y 389.347,Z 521.634,A -85,B 0,C 180,E1 -11619.875,E2 -11619.875} C_VEL
LIN {X 0,Y 389.814,Z 513.637,A -85,B 0,C 180,E1 -11621.44,E2 -11621.44} C_VEL
LIN {X 0,Y 390.379,Z 505.486,A -85,B 0,C 180,E1 -11622.741,E2 -11622.741} C_VEL
LIN {X 0,Y 391.036,Z 495.147,A -85,B 0,C 180,E1 -11624.09,E2 -11624.09} C_VEL
LIN {X 0,Y 391.859,Z 484.504,A -85,B 0,C 180,E1 -11625.207,E2 -11625.207} C_VEL
LIN {X 0,Y 392.679,Z 473.725,A -85,B 0,C 180,E1 -11626.107,E2 -11626.107} C_VEL
LIN {X 0,Y 391.999,Z 460.438,A -85,B 0,C 180,E1 -11627.003,E2 -11627.003} C_VEL
LIN {X 0,Y 390.931,Z 447.291,A -85,B 0,C 180,E1 -11627.671,E2 -11627.671} C_VEL
LIN {X 0,Y 389.543,Z 433.945,A -85,B 0,C 180,E1 -11628.133,E2 -11628.133} C_VEL
LIN {X 0,Y 389.397,Z 432.037,A -85,B 0,C 180,E1 -11628.209,E2 -11628.209} C_VEL
LIN {X 0,Y 389.793,Z 420.591,A -85,B 0,C 180,E1 -11631.693,E2 -11631.693} C_VEL
LIN {X 0,Y 390.29,Z 409.702,A -85,B 0,C 180,E1 -11635.036,E2 -11635.036} C_VEL
LIN {X 0,Y 390.957,Z 398.27,A -85,B 0,C 180,E1 -11638.583,E2 -11638.583} C_VEL
LIN {X 0,Y 391.667,Z 387.616,A -85,B 0,C 180,E1 -11641.954,E2 -11641.954} C_VEL
LIN {X 0,Y 392.609,Z 376.468,A -85,B 0,C 180,E1 -11645.576,E2 -11645.576} C_VEL
LIN {X 0,Y 392.85,Z 372.596,A -85,B 0,C 180,E1 -11646.87,E2 -11646.87} C_VEL
LIN {X 0,Y 391.54,Z 364.367,A -85,B 0,C 180,E1 -11649.831,E2 -11649.831} C_VEL
LIN {X 0,Y 390.103,Z 356.894,A -85,B 0,C 180,E1 -11652.753,E2 -11652.753} C_VEL
LIN {X 0,Y 390.059,Z 356.902,A -85,B 0,C 180,E1 -11656.114,E2 -11656.114} C_VEL
LIN {X 0,Y 390.06,Z 356.896,A -85,B 0,C 180,E1 -11659.561,E2 -11659.561} C_VEL
LIN {X 0,Y 390.048,Z 356.899,A -85,B 0,C 180,E1 -11662.45,E2 -11662.45} C_VEL
LIN {X 0,Y 390.072,Z 356.894,A -85,B 0,C 180,E1 -11665.976,E2 -11665.976} C_VEL
LIN {X 0,Y 390.051,Z 356.896,A -85,B 0,C 180,E1 -11669.869,E2 -11669.869} C_VEL
LIN {X 0,Y 390.118,Z 356.89,A -85,B 0,C 180,E1 -11673.232,E2 -11673.232} C_VEL
LIN {X 0,Y 390.112,Z 356.894,A -85,B 0,C 180,E1 -11676.751,E2 -11676.751} C_VEL
LIN {X 0,Y 390.109,Z 356.89,A -85,B 0,C 180,E1 -11679.983,E2 -11679.983} C_VEL
LIN {X 0,Y 390.143,Z 356.885,A -85,B 0,C 180,E1 -11683.249,E2 -11683.249} C_VEL
LIN {X 0,Y 390.2,Z 356.883,A -85,B 0,C 180,E1 -11686.562,E2 -11686.562} C_VEL
LIN {X 0,Y 390.21,Z 356.88,A -85,B 0,C 180,E1 -11690.672,E2 -11690.672} C_VEL
LIN {X 0,Y 390.325,Z 356.865,A -85,B 0,C 180,E1 -11692.759,E2 -11692.759} C_VEL
LIN {X 0,Y 390.231,Z 356.876,A -85,B 0,C 180,E1 -11694.834,E2 -11694.834} C_VEL
LIN {X 0,Y 390.424,Z 356.853,A -85,B 0,C 180,E1 -11697.937,E2 -11697.937} C_VEL
LIN {X 0,Y 390.556,Z 356.837,A -85,B 0,C 180,E1 -11700,E2 -11700} C_VEL
LIN {X 0,Y 390.315,Z 356.864,A -85,B 0,C 180,E1 -11703.097,E2 -11703.097} C_VEL
LIN {X 0,Y 390.315,Z 356.864,A -85,B 0,C 180,E1 -11706.655,E2 -11706.655} C_VEL
LIN {X 0,Y 390.211,Z 356.877,A -85,B 0,C 180,E1 -11709.329,E2 -11709.329} C_VEL
LIN {X 0,Y 390.201,Z 356.879,A -85,B 0,C 180,E1 -11713.439,E2 -11713.439} C_VEL
LIN {X 0,Y 390.155,Z 356.885,A -85,B 0,C 180,E1 -11717.308,E2 -11717.308} C_VEL
LIN {X 0,Y 390.094,Z 356.892,A -85,B 0,C 180,E1 -11720.47,E2 -11720.47} C_VEL
LIN {X 0,Y 390.096,Z 356.893,A -85,B 0,C 180,E1 -11723.351,E2 -11723.351} C_VEL
LIN {X 0,Y 390.12,Z 356.888,A -85,B 0,C 180,E1 -11726.768,E2 -11726.768} C_VEL
LIN {X 0,Y 390.045,Z 356.898,A -85,B 0,C 180,E1 -11730.3,E2 -11730.3} C_VEL
LIN {X 0,Y 390.074,Z 356.896,A -85,B 0,C 180,E1 -11734.025,E2 -11734.025} C_VEL
LIN {X 0,Y 390.05,Z 356.901,A -85,B 0,C 180,E1 -11737.551,E2 -11737.551} C_VEL
LIN {X 0,Y 390.063,Z 356.896,A -85,B 0,C 180,E1 -11740.821,E2 -11740.821} C_VEL
LIN {X 0,Y 390.061,Z 356.897,A -85,B 0,C 180,E1 -11743.886,E2 -11743.886} C_VEL
LIN {X 0,Y 390.063,Z 356.896,A -85,B 0,C 180,E1 -11746.789,E2 -11746.789} C_VEL
LIN {X 0,Y 390.062,Z 356.899,A -85,B 0,C 180,E1 -11749.56,E2 -11749.56} C_VEL
LIN {X 0,Y 390.049,Z 356.897,A -85,B 0,C 180,E1 -11752.449,E2 -11752.449} C_VEL
LIN {X 0,Y 390.074,Z 356.894,A -85,B 0,C 180,E1 -11755.975,E2 -11755.975} C_VEL
LIN {X 0,Y 390.053,Z 356.896,A -85,B 0,C 180,E1 -11759.869,E2 -11759.869} C_VEL
LIN {X 0,Y 390.12,Z 356.892,A -85,B 0,C 180,E1 -11763.231,E2 -11763.231} C_VEL
LIN {X 0,Y 390.113,Z 356.893,A -85,B 0,C 180,E1 -11766.75,E2 -11766.75} C_VEL
LIN {X 0,Y 390.11,Z 356.889,A -85,B 0,C 180,E1 -11769.983,E2 -11769.983} C_VEL
LIN {X 0,Y 390.144,Z 356.887,A -85,B 0,C 180,E1 -11773.248,E2 -11773.248} C_VEL
LIN {X 0,Y 390.2,Z 356.883,A -85,B 0,C 180,E1 -11776.561,E2 -11776.561} C_VEL
LIN {X 0,Y 390.21,Z 356.881,A -85,B 0,C 180,E1 -11780.474,E2 -11780.474} C_VEL
LIN {X 0,Y 394.273,Z 370.591,A -85,B 0,C 180,E1 -11781.406,E2 -11781.406} C_VEL
LIN {X 0,Y 394.873,Z 373.78,A -85,B 0,C 180,E1 -11781.647,E2 -11781.647} C_VEL
LIN {X 0,Y 394.238,Z 385.893,A -85,B 0,C 180,E1 -11782.573,E2 -11782.573} C_VEL
LIN {X 0,Y 393.46,Z 397.433,A -85,B 0,C 180,E1 -11783.718,E2 -11783.718} C_VEL
LIN {X 0,Y 392.838,Z 406.721,A -85,B 0,C 180,E1 -11784.867,E2 -11784.867} C_VEL
LIN {X 0,Y 392.17,Z 415.218,A -85,B 0,C 180,E1 -11786.146,E2 -11786.146} C_VEL
LIN {X 0,Y 391.442,Z 423.483,A -85,B 0,C 180,E1 -11787.684,E2 -11787.684} C_VEL
LIN {X 0,Y 390.897,Z 429.149,A -85,B 0,C 180,E1 -11788.969,E2 -11788.969} C_VEL
LIN {X 0,Y 390.476,Z 434.653,A -85,B 0,C 180,E1 -11790.515,E2 -11790.515} C_VEL
LIN {X 0,Y 390.147,Z 438.995,A -85,B 0,C 180,E1 -11792.064,E2 -11792.064} C_VEL
LIN {X 0,Y 389.881,Z 441.309,A -85,B 0,C 180,E1 -11793.099,E2 -11793.099} C_VEL
LIN {X 0,Y 389.779,Z 443.188,A -85,B 0,C 180,E1 -11794.135,E2 -11794.135} C_VEL
LIN {X 0,Y 389.796,Z 444.628,A -85,B 0,C 180,E1 -11795.171,E2 -11795.171} C_VEL
LIN {X 0,Y 389.749,Z 446.303,A -85,B 0,C 180,E1 -11797.251,E2 -11797.251} C_VEL
LIN {X 0,Y 389.708,Z 446.586,A -85,B 0,C 180,E1 -11798.294,E2 -11798.294} C_VEL
LIN {X 0,Y 389.732,Z 446.458,A -85,B 0,C 180,E1 -11799.339,E2 -11799.339} C_VEL
LIN {X 0,Y 389.881,Z 444.992,A -85,B 0,C 180,E1 -11801.436,E2 -11801.436} C_VEL
LIN {X 0,Y 390.136,Z 443.663,A -85,B 0,C 180,E1 -11802.483,E2 -11802.483} C_VEL
LIN {X 0,Y 390.457,Z 440.841,A -85,B 0,C 180,E1 -11804.062,E2 -11804.062} C_VEL
LIN {X 0,Y 390.917,Z 436.971,A -85,B 0,C 180,E1 -11805.644,E2 -11805.644} C_VEL
LIN {X 0,Y 391.508,Z 431.931,A -85,B 0,C 180,E1 -11807.228,E2 -11807.228} C_VEL
LIN {X 0,Y 392.211,Z 425.512,A -85,B 0,C 180,E1 -11808.816,E2 -11808.816} C_VEL
LIN {X 0,Y 393.124,Z 417.452,A -85,B 0,C 180,E1 -11810.401,E2 -11810.401} C_VEL
LIN {X 0,Y 394.006,Z 408.696,A -85,B 0,C 180,E1 -11811.794,E2 -11811.794} C_VEL
LIN {X 0,Y 394.569,Z 402.473,A -85,B 0,C 180,E1 -11812.619,E2 -11812.619} C_VEL
LIN {X 0,Y 394.395,Z 396.526,A -85,B 0,C 180,E1 -11813.355,E2 -11813.355} C_VEL
LIN {X 0,Y 393.141,Z 390.541,A -85,B 0,C 180,E1 -11814.078,E2 -11814.078} C_VEL
LIN {X 0,Y 391.404,Z 384.389,A -85,B 0,C 180,E1 -11814.768,E2 -11814.768} C_VEL
LIN {X 0,Y 389.785,Z 377.922,A -85,B 0,C 180,E1 -11815.402,E2 -11815.402} C_VEL
LIN {X 0,Y 386.975,Z 368.688,A -85,B 0,C 180,E1 -11816.216,E2 -11816.216} C_VEL
LIN {X 0,Y 383.083,Z 357.77,A -85,B 0,C 180,E1 -11817.058,E2 -11817.058} C_VEL
LIN {X 0,Y 382.984,Z 357.78,A -85,B 0,C 180,E1 -11820.918,E2 -11820.918} C_VEL
LIN {X 0,Y 383.018,Z 357.778,A -85,B 0,C 180,E1 -11824.667,E2 -11824.667} C_VEL
LIN {X 0,Y 383,Z 357.778,A -85,B 0,C 180,E1 -11827.903,E2 -11827.903} C_VEL
LIN {X 0,Y 382.985,Z 357.781,A -85,B 0,C 180,E1 -11831.346,E2 -11831.346} C_VEL
LIN {X 0,Y 382.997,Z 357.778,A -85,B 0,C 180,E1 -11834.303,E2 -11834.303} C_VEL
LIN {X 0,Y 383.038,Z 357.772,A -85,B 0,C 180,E1 -11837.243,E2 -11837.243} C_VEL
LIN {X 0,Y 383.021,Z 357.774,A -85,B 0,C 180,E1 -11840.411,E2 -11840.411} C_VEL
LIN {X 0,Y 383.025,Z 357.772,A -85,B 0,C 180,E1 -11844.044,E2 -11844.044} C_VEL
LIN {X 0,Y 383.035,Z 357.765,A -85,B 0,C 180,E1 -11847.852,E2 -11847.852} C_VEL
LIN {X 0,Y 383.061,Z 357.757,A -85,B 0,C 180,E1 -11851.72,E2 -11851.72} C_VEL
LIN {X 0,Y 383.05,Z 357.771,A -85,B 0,C 180,E1 -11855.039,E2 -11855.039} C_VEL
LIN {X 0,Y 382.99,Z 357.778,A -85,B 0,C 180,E1 -11858.468,E2 -11858.468} C_VEL
LIN {X 0,Y 383.086,Z 357.76,A -85,B 0,C 180,E1 -11861.827,E2 -11861.827} C_VEL
LIN {X 0,Y 383.109,Z 357.765,A -85,B 0,C 180,E1 -11865.118,E2 -11865.118} C_VEL
LIN {X 0,Y 383.106,Z 357.766,A -85,B 0,C 180,E1 -11868.358,E2 -11868.358} C_VEL
LIN {X 0,Y 383.3,Z 357.74,A -85,B 0,C 180,E1 -11871.932,E2 -11871.932} C_VEL
LIN {X 0,Y 383.197,Z 357.745,A -85,B 0,C 180,E1 -11874.738,E2 -11874.738} C_VEL
LIN {X 0,Y 383.385,Z 357.73,A -85,B 0,C 180,E1 -11877.899,E2 -11877.899} C_VEL
LIN {X 0,Y 383.518,Z 357.705,A -85,B 0,C 180,E1 -11880,E2 -11880} C_VEL
LIN {X 0,Y 383.249,Z 357.748,A -85,B 0,C 180,E1 -11883.153,E2 -11883.153} C_VEL
LIN {X 0,Y 383.284,Z 357.741,A -85,B 0,C 180,E1 -11886.316,E2 -11886.316} C_VEL
LIN {X 0,Y 383.256,Z 357.745,A -85,B 0,C 180,E1 -11888.436,E2 -11888.436} C_VEL
LIN {X 0,Y 383.094,Z 357.766,A -85,B 0,C 180,E1 -11891.642,E2 -11891.642} C_VEL
LIN {X 0,Y 383.106,Z 357.763,A -85,B 0,C 180,E1 -11894.882,E2 -11894.882} C_VEL
LIN {X 0,Y 383.085,Z 357.765,A -85,B 0,C 180,E1 -11898.172,E2 -11898.172} C_VEL
LIN {X 0,Y 382.989,Z 357.781,A -85,B 0,C 180,E1 -11901.531,E2 -11901.531} C_VEL
LIN {X 0,Y 383.048,Z 357.775,A -85,B 0,C 180,E1 -11904.96,E2 -11904.96} C_VEL
LIN {X 0,Y 383.046,Z 357.775,A -85,B 0,C 180,E1 -11908.492,E2 -11908.492} C_VEL
LIN {X 0,Y 383.008,Z 357.779,A -85,B 0,C 180,E1 -11912.15,E2 -11912.15} C_VEL
LIN {X 0,Y 383.015,Z 357.777,A -85,B 0,C 180,E1 -11914.668,E2 -11914.668} C_VEL
LIN {X 0,Y 383,Z 357.771,A -85,B 0,C 180,E1 -11917.905,E2 -11917.905} C_VEL
LIN {X 0,Y 383.043,Z 357.765,A -85,B 0,C 180,E1 -11921.34,E2 -11921.34} C_VEL
LIN {X 0,Y 383.074,Z 357.848,A -85,B 0,C 180,E1 -11924.771,E2 -11924.771} C_VEL
LIN {X 0,Y 384.493,Z 364.915,A -85,B 0,C 180,E1 -11927.879,E2 -11927.879} C_VEL
LIN {X 0,Y 385.929,Z 372.541,A -85,B 0,C 180,E1 -11931.003,E2 -11931.003} C_VEL
LIN {X 0,Y 386.59,Z 376.324,A -85,B 0,C 180,E1 -11932.484,E2 -11932.484} C_VEL
LIN {X 0,Y 386.466,Z 379.866,A -85,B 0,C 180,E1 -11933.771,E2 -11933.771} C_VEL
LIN {X 0,Y 385.262,Z 390.695,A -85,B 0,C 180,E1 -11937.537,E2 -11937.537} C_VEL
LIN {X 0,Y 384.306,Z 400.917,A -85,B 0,C 180,E1 -11940.973,E2 -11940.973} C_VEL
LIN {X 0,Y 383.52,Z 411.642,A -85,B 0,C 180,E1 -11944.493,E2 -11944.493} C_VEL
LIN {X 0,Y 382.883,Z 422.202,A -85,B 0,C 180,E1 -11947.897,E2 -11947.897} C_VEL
LIN {X 0,Y 382.497,Z 430.363,A -85,B 0,C 180,E1 -11950.496,E2 -11950.496} C_VEL
LIN {X 0,Y 384.771,Z 444.431,A -85,B 0,C 180,E1 -11951.058,E2 -11951.058} C_VEL
LIN {X 0,Y 386.124,Z 457.097,A -85,B 0,C 180,E1 -11951.737,E2 -11951.737} C_VEL
LIN {X 0,Y 386.549,Z 469.047,A -85,B 0,C 180,E1 -11952.544,E2 -11952.544} C_VEL
LIN {X 0,Y 386.568,Z 477.421,A -85,B 0,C 180,E1 -11953.226,E2 -11953.226} C_VEL
LIN {X 0,Y 385.409,Z 488.329,A -85,B 0,C 180,E1 -11954.262,E2 -11954.262} C_VEL
LIN {X 0,Y 384.464,Z 497.906,A -85,B 0,C 180,E1 -11955.394,E2 -11955.394} C_VEL
LIN {X 0,Y 383.689,Z 507.353,A -85,B 0,C 180,E1 -11956.765,E2 -11956.765} C_VEL
LIN {X 0,Y 382.933,Z 514.884,A -85,B 0,C 180,E1 -11958.085,E2 -11958.085} C_VEL
LIN {X 0,Y 382.316,Z 522.336,A -85,B 0,C 180,E1 -11959.676,E2 -11959.676} C_VEL
LIN {X 0,Y 382.052,Z 529.236,A -85,B 0,C 180,E1 -11961.538,E2 -11961.538} C_VEL
LIN {X 0,Y 382.005,Z 534.612,A -85,B 0,C 180,E1 -11963.452,E2 -11963.452} C_VEL
LIN {X 0,Y 382.032,Z 537.346,A -85,B 0,C 180,E1 -11964.723,E2 -11964.723} C_VEL
LIN {X 0,Y 382.177,Z 539.118,A -85,B 0,C 180,E1 -11965.782,E2 -11965.782} C_VEL
LIN {X 0,Y 382.277,Z 540.474,A -85,B 0,C 180,E1 -11966.839,E2 -11966.839} C_VEL
LIN {X 0,Y 382.208,Z 541.405,A -85,B 0,C 180,E1 -11967.893,E2 -11967.893} C_VEL
LIN {X 0,Y 382.232,Z 541.904,A -85,B 0,C 180,E1 -11968.947,E2 -11968.947} C_VEL
LIN {X 0,Y 382.288,Z 541.993,A -85,B 0,C 180,E1 -11970.001,E2 -11970.001} C_VEL
LIN {X 0,Y 382.259,Z 541.674,A -85,B 0,C 180,E1 -11971.054,E2 -11971.054} C_VEL
LIN {X 0,Y 382.25,Z 540.958,A -85,B 0,C 180,E1 -11972.108,E2 -11972.108} C_VEL
LIN {X 0,Y 382.299,Z 539.804,A -85,B 0,C 180,E1 -11973.162,E2 -11973.162} C_VEL
LIN {X 0,Y 382.192,Z 537.246,A -85,B 0,C 180,E1 -11974.747,E2 -11974.747} C_VEL
LIN {X 0,Y 382.09,Z 532.746,A -85,B 0,C 180,E1 -11976.658,E2 -11976.658} C_VEL
LIN {X 0,Y 382.121,Z 527.023,A -85,B 0,C 180,E1 -11978.462,E2 -11978.462} C_VEL
LIN {X 0,Y 382.291,Z 520.565,A -85,B 0,C 180,E1 -11980.059,E2 -11980.059} C_VEL
LIN {X 0,Y 382.79,Z 512.506,A -85,B 0,C 180,E1 -11981.652,E2 -11981.652} C_VEL
LIN {X 0,Y 383.416,Z 504.308,A -85,B 0,C 180,E1 -11982.977,E2 -11982.977} C_VEL
LIN {X 0,Y 384.046,Z 494.732,A -85,B 0,C 180,E1 -11984.25,E2 -11984.25} C_VEL
LIN {X 0,Y 384.847,Z 484.511,A -85,B 0,C 180,E1 -11985.356,E2 -11985.356} C_VEL
LIN {X 0,Y 385.674,Z 473.999,A -85,B 0,C 180,E1 -11986.271,E2 -11986.271} C_VEL
LIN {X 0,Y 385.086,Z 462.018,A -85,B 0,C 180,E1 -11987.126,E2 -11987.126} C_VEL
LIN {X 0,Y 384.061,Z 448.527,A -85,B 0,C 180,E1 -11987.859,E2 -11987.859} C_VEL
LIN {X 0,Y 382.794,Z 435.485,A -85,B 0,C 180,E1 -11988.361,E2 -11988.361} C_VEL
LIN {X 0,Y 382.303,Z 431.235,A -85,B 0,C 180,E1 -11988.489,E2 -11988.489} C_VEL
LIN {X 0,Y 382.765,Z 419.612,A -85,B 0,C 180,E1 -11992.112,E2 -11992.112} C_VEL
LIN {X 0,Y 383.266,Z 408.788,A -85,B 0,C 180,E1 -11995.508,E2 -11995.508} C_VEL
LIN {X 0,Y 383.966,Z 397.727,A -85,B 0,C 180,E1 -11999.016,E2 -11999.016} C_VEL
LIN {X 0,Y 384.736,Z 387.2,A -85,B 0,C 180,E1 -12002.428,E2 -12002.428} C_VEL
LIN {X 0,Y 385.77,Z 375.883,A -85,B 0,C 180,E1 -12006.201,E2 -12006.201} C_VEL
LIN {X 0,Y 385.86,Z 373.708,A -85,B 0,C 180,E1 -12006.947,E2 -12006.947} C_VEL
LIN {X 0,Y 384.574,Z 365.747,A -85,B 0,C 180,E1 -12009.866,E2 -12009.866} C_VEL
LIN {X 0,Y 383.057,Z 357.772,A -85,B 0,C 180,E1 -12013.014,E2 -12013.014} C_VEL
LIN {X 0,Y 383.002,Z 357.779,A -85,B 0,C 180,E1 -12015.79,E2 -12015.79} C_VEL
LIN {X 0,Y 382.992,Z 357.78,A -85,B 0,C 180,E1 -12018.796,E2 -12018.796} C_VEL
LIN {X 0,Y 383.004,Z 357.774,A -85,B 0,C 180,E1 -12022.097,E2 -12022.097} C_VEL
LIN {X 0,Y 383.022,Z 357.774,A -85,B 0,C 180,E1 -12025.333,E2 -12025.333} C_VEL
LIN {X 0,Y 382.988,Z 357.78,A -85,B 0,C 180,E1 -12029.082,E2 -12029.082} C_VEL
LIN {X 0,Y 383.061,Z 357.772,A -85,B 0,C 180,E1 -12032.699,E2 -12032.699} C_VEL
LIN {X 0,Y 383.057,Z 357.77,A -85,B 0,C 180,E1 -12035.04,E2 -12035.04} C_VEL
LIN {X 0,Y 382.998,Z 357.779,A -85,B 0,C 180,E1 -12038.469,E2 -12038.469} C_VEL
LIN {X 0,Y 383.068,Z 357.766,A -85,B 0,C 180,E1 -12041.827,E2 -12041.827} C_VEL
LIN {X 0,Y 383.116,Z 357.761,A -85,B 0,C 180,E1 -12045.119,E2 -12045.119} C_VEL
LIN {X 0,Y 383.103,Z 357.767,A -85,B 0,C 180,E1 -12048.358,E2 -12048.358} C_VEL
LIN {X 0,Y 383.31,Z 357.738,A -85,B 0,C 180,E1 -12051.933,E2 -12051.933} C_VEL
LIN {X 0,Y 383.204,Z 357.752,A -85,B 0,C 180,E1 -12054.739,E2 -12054.739} C_VEL
LIN {X 0,Y 383.391,Z 357.729,A -85,B 0,C 180,E1 -12057.899,E2 -12057.899} C_VEL
LIN {X 0,Y 383.526,Z 357.713,A -85,B 0,C 180,E1 -12060,E2 -12060} C_VEL
LIN {X 0,Y 383.252,Z 357.743,A -85,B 0,C 180,E1 -12063.154,E2 -12063.154} C_VEL
LIN {X 0,Y 383.275,Z 357.741,A -85,B 0,C 180,E1 -12066.65,E2 -12066.65} C_VEL
LIN {X 0,Y 383.266,Z 357.744,A -85,B 0,C 180,E1 -12068.436,E2 -12068.436} C_VEL
LIN {X 0,Y 383.104,Z 357.765,A -85,B 0,C 180,E1 -12071.642,E2 -12071.642} C_VEL
LIN {X 0,Y 383.116,Z 357.76,A -85,B 0,C 180,E1 -12074.882,E2 -12074.882} C_VEL
LIN {X 0,Y 383.096,Z 357.766,A -85,B 0,C 180,E1 -12078.172,E2 -12078.172} C_VEL
LIN {X 0,Y 382.999,Z 357.778,A -85,B 0,C 180,E1 -12081.531,E2 -12081.531} C_VEL
LIN {X 0,Y 383.058,Z 357.768,A -85,B 0,C 180,E1 -12084.96,E2 -12084.96} C_VEL
LIN {X 0,Y 383.036,Z 357.771,A -85,B 0,C 180,E1 -12088.27,E2 -12088.27} C_VEL
LIN {X 0,Y 383.016,Z 357.774,A -85,B 0,C 180,E1 -12092.15,E2 -12092.15} C_VEL
LIN {X 0,Y 383.024,Z 357.772,A -85,B 0,C 180,E1 -12094.668,E2 -12094.668} C_VEL
LIN {X 0,Y 383.006,Z 357.776,A -85,B 0,C 180,E1 -12097.904,E2 -12097.904} C_VEL
LIN {X 0,Y 382.991,Z 357.781,A -85,B 0,C 180,E1 -12101.347,E2 -12101.347} C_VEL
LIN {X 0,Y 383.002,Z 357.774,A -85,B 0,C 180,E1 -12104.303,E2 -12104.303} C_VEL
LIN {X 0,Y 383.016,Z 357.778,A -85,B 0,C 180,E1 -12107.24,E2 -12107.24} C_VEL
LIN {X 0,Y 383.021,Z 357.772,A -85,B 0,C 180,E1 -12110.413,E2 -12110.413} C_VEL
LIN {X 0,Y 383.031,Z 357.771,A -85,B 0,C 180,E1 -12114.044,E2 -12114.044} C_VEL
LIN {X 0,Y 382.993,Z 357.777,A -85,B 0,C 180,E1 -12117.578,E2 -12117.578} C_VEL
LIN {X 0,Y 382.998,Z 357.775,A -85,B 0,C 180,E1 -12120.3,E2 -12120.3} C_VEL
LIN {X 0,Y 383.087,Z 357.764,A -85,B 0,C 180,E1 -12124.02,E2 -12124.02} C_VEL
LIN {X 0,Y 383.015,Z 357.775,A -85,B 0,C 180,E1 -12127.335,E2 -12127.335} C_VEL
LIN {X 0,Y 383.067,Z 357.771,A -85,B 0,C 180,E1 -12130.716,E2 -12130.716} C_VEL
LIN {X 0,Y 383.087,Z 357.764,A -85,B 0,C 180,E1 -12134.026,E2 -12134.026} C_VEL
LIN {X 0,Y 383.143,Z 357.758,A -85,B 0,C 180,E1 -12137.283,E2 -12137.283} C_VEL
LIN {X 0,Y 383.17,Z 357.757,A -85,B 0,C 180,E1 -12140.198,E2 -12140.198} C_VEL
LIN {X 0,Y 387.027,Z 370.655,A -85,B 0,C 180,E1 -12141.081,E2 -12141.081} C_VEL
LIN {X 0,Y 387.964,Z 374.243,A -85,B 0,C 180,E1 -12141.366,E2 -12141.366} C_VEL
LIN {X 0,Y 387.397,Z 386.448,A -85,B 0,C 180,E1 -12142.31,E2 -12142.31} C_VEL
LIN {X 0,Y 386.698,Z 396.891,A -85,B 0,C 180,E1 -12143.346,E2 -12143.346} C_VEL
LIN {X 0,Y 386.008,Z 406.425,A -85,B 0,C 180,E1 -12144.514,E2 -12144.514} C_VEL
LIN {X 0,Y 385.318,Z 415.111,A -85,B 0,C 180,E1 -12145.815,E2 -12145.815} C_VEL
LIN {X 0,Y 384.543,Z 423.611,A -85,B 0,C 180,E1 -12147.38,E2 -12147.38} C_VEL
LIN {X 0,Y 383.882,Z 430.401,A -85,B 0,C 180,E1 -12148.95,E2 -12148.95} C_VEL
LIN {X 0,Y 383.448,Z 435.83,A -85,B 0,C 180,E1 -12150.524,E2 -12150.524} C_VEL
LIN {X 0,Y 383.101,Z 440.104,A -85,B 0,C 180,E1 -12152.102,E2 -12152.102} C_VEL
LIN {X 0,Y 382.828,Z 442.386,A -85,B 0,C 180,E1 -12153.156,E2 -12153.156} C_VEL
LIN {X 0,Y 382.737,Z 444.229,A -85,B 0,C 180,E1 -12154.211,E2 -12154.211} C_VEL
LIN {X 0,Y 382.743,Z 445.61,A -85,B 0,C 180,E1 -12155.267,E2 -12155.267} C_VEL
LIN {X 0,Y 382.69,Z 447.226,A -85,B 0,C 180,E1 -12157.385,E2 -12157.385} C_VEL
LIN {X 0,Y 382.677,Z 447.471,A -85,B 0,C 180,E1 -12158.448,E2 -12158.448} C_VEL
LIN {X 0,Y 382.759,Z 446.717,A -85,B 0,C 180,E1 -12160.58,E2 -12160.58} C_VEL
LIN {X 0,Y 382.888,Z 445.76,A -85,B 0,C 180,E1 -12161.648,E2 -12161.648} C_VEL
LIN {X 0,Y 383.152,Z 444.386,A -85,B 0,C 180,E1 -12162.715,E2 -12162.715} C_VEL
LIN {X 0,Y 383.52,Z 441.504,A -85,B 0,C 180,E1 -12164.322,E2 -12164.322} C_VEL
LIN {X 0,Y 384.014,Z 437.561,A -85,B 0,C 180,E1 -12165.933,E2 -12165.933} C_VEL
LIN {X 0,Y 384.771,Z 431.424,A -85,B 0,C 180,E1 -12167.814,E2 -12167.814} C_VEL
LIN {X 0,Y 385.566,Z 424.686,A -85,B 0,C 180,E1 -12169.429,E2 -12169.429} C_VEL
LIN {X 0,Y 386.408,Z 417.752,A -85,B 0,C 180,E1 -12170.772,E2 -12170.772} C_VEL
LIN {X 0,Y 387.254,Z 409.514,A -85,B 0,C 180,E1 -12172.094,E2 -12172.094} C_VEL
LIN {X 0,Y 388.111,Z 400.022,A -85,B 0,C 180,E1 -12173.335,E2 -12173.335} C_VEL
LIN {X 0,Y 389.126,Z 388.352,A -85,B 0,C 180,E1 -12174.544,E2 -12174.544} C_VEL
LIN {X 0,Y 389.785,Z 377.922,A -85,B 0,C 180,E1 -12175.402,E2 -12175.402} C_VEL
LIN {X 0,Y 388.379,Z 374.914,A -85,B 0,C 180,E1 -12175.716,E2 -12175.716} C_VEL
LIN {X 0,Y 384.24,Z 371.026,A -85,B 0,C 180,E1 -12176.251,E2 -12176.251} C_VEL
LIN {X 0,Y 379.841,Z 367.149,A -85,B 0,C 180,E1 -12176.777,E2 -12176.777} C_VEL
LIN {X 0,Y 378.017,Z 364.123,A -85,B 0,C 180,E1 -12177.069,E2 -12177.069} C_VEL
LIN {X 0,Y 376.021,Z 358.65,A -85,B 0,C 180,E1 -12177.485,E2 -12177.485} C_VEL
LIN {X 0,Y 375.959,Z 358.657,A -85,B 0,C 180,E1 -12181.561,E2 -12181.561} C_VEL
LIN {X 0,Y 375.958,Z 358.66,A -85,B 0,C 180,E1 -12185.414,E2 -12185.414} C_VEL
LIN {X 0,Y 375.974,Z 358.653,A -85,B 0,C 180,E1 -12188.27,E2 -12188.27} C_VEL
LIN {X 0,Y 375.935,Z 358.657,A -85,B 0,C 180,E1 -12191.6,E2 -12191.6} C_VEL
LIN {X 0,Y 375.928,Z 358.661,A -85,B 0,C 180,E1 -12195.267,E2 -12195.267} C_VEL
LIN {X 0,Y 375.959,Z 358.658,A -85,B 0,C 180,E1 -12198.394,E2 -12198.394} C_VEL
LIN {X 0,Y 375.977,Z 358.655,A -85,B 0,C 180,E1 -12201.728,E2 -12201.728} C_VEL
LIN {X 0,Y 375.978,Z 358.654,A -85,B 0,C 180,E1 -12205.332,E2 -12205.332} C_VEL
LIN {X 0,Y 375.974,Z 358.638,A -85,B 0,C 180,E1 -12208.439,E2 -12208.439} C_VEL
LIN {X 0,Y 376,Z 358.64,A -85,B 0,C 180,E1 -12212.141,E2 -12212.141} C_VEL
LIN {X 0,Y 376.004,Z 358.649,A -85,B 0,C 180,E1 -12214.538,E2 -12214.538} C_VEL
LIN {X 0,Y 375.96,Z 358.651,A -85,B 0,C 180,E1 -12218.045,E2 -12218.045} C_VEL
LIN {X 0,Y 376.021,Z 358.641,A -85,B 0,C 180,E1 -12221.473,E2 -12221.473} C_VEL
LIN {X 0,Y 376.057,Z 358.643,A -85,B 0,C 180,E1 -12224.832,E2 -12224.832} C_VEL
LIN {X 0,Y 376.057,Z 358.644,A -85,B 0,C 180,E1 -12228.137,E2 -12228.137} C_VEL
LIN {X 0,Y 376.254,Z 358.618,A -85,B 0,C 180,E1 -12231.877,E2 -12231.877} C_VEL
LIN {X 0,Y 376.169,Z 358.62,A -85,B 0,C 180,E1 -12234.64,E2 -12234.64} C_VEL
LIN {X 0,Y 376.351,Z 358.606,A -85,B 0,C 180,E1 -12237.859,E2 -12237.859} C_VEL
LIN {X 0,Y 376.487,Z 358.58,A -85,B 0,C 180,E1 -12240,E2 -12240} C_VEL
LIN {X 0,Y 376.187,Z 358.628,A -85,B 0,C 180,E1 -12243.213,E2 -12243.213} C_VEL
LIN {X 0,Y 376.243,Z 358.618,A -85,B 0,C 180,E1 -12246.435,E2 -12246.435} C_VEL
LIN {X 0,Y 376.201,Z 358.623,A -85,B 0,C 180,E1 -12248.595,E2 -12248.595} C_VEL
LIN {X 0,Y 376.046,Z 358.644,A -85,B 0,C 180,E1 -12251.863,E2 -12251.863} C_VEL
LIN {X 0,Y 376.054,Z 358.642,A -85,B 0,C 180,E1 -12255.167,E2 -12255.167} C_VEL
LIN {X 0,Y 376.02,Z 358.648,A -85,B 0,C 180,E1 -12258.526,E2 -12258.526} C_VEL
LIN {X 0,Y 375.959,Z 358.656,A -85,B 0,C 180,E1 -12261.954,E2 -12261.954} C_VEL
LIN {X 0,Y 376.002,Z 358.652,A -85,B 0,C 180,E1 -12265.461,E2 -12265.461} C_VEL
LIN {X 0,Y 375.973,Z 358.657,A -85,B 0,C 180,E1 -12269.079,E2 -12269.079} C_VEL
LIN {X 0,Y 375.948,Z 358.658,A -85,B 0,C 180,E1 -12272.829,E2 -12272.829} C_VEL
LIN {X 0,Y 375.955,Z 358.655,A -85,B 0,C 180,E1 -12275.416,E2 -12275.416} C_VEL
LIN {X 0,Y 375.975,Z 358.643,A -85,B 0,C 180,E1 -12278.272,E2 -12278.272} C_VEL
LIN {X 0,Y 375.986,Z 358.643,A -85,B 0,C 180,E1 -12281.611,E2 -12281.611} C_VEL
LIN {X 0,Y 376.03,Z 358.664,A -85,B 0,C 180,E1 -12284.281,E2 -12284.281} C_VEL
LIN {X 0,Y 377.642,Z 366.828,A -85,B 0,C 180,E1 -12287.936,E2 -12287.936} C_VEL
LIN {X 0,Y 378.98,Z 373.962,A -85,B 0,C 180,E1 -12290.913,E2 -12290.913} C_VEL
LIN {X 0,Y 379.681,Z 378.564,A -85,B 0,C 180,E1 -12292.744,E2 -12292.744} C_VEL
LIN {X 0,Y 379.019,Z 384.553,A -85,B 0,C 180,E1 -12294.914,E2 -12294.914} C_VEL
LIN {X 0,Y 377.923,Z 395.105,A -85,B 0,C 180,E1 -12298.622,E2 -12298.622} C_VEL
LIN {X 0,Y 376.977,Z 405.683,A -85,B 0,C 180,E1 -12302.221,E2 -12302.221} C_VEL
LIN {X 0,Y 376.098,Z 417.944,A -85,B 0,C 180,E1 -12306.297,E2 -12306.297} C_VEL
LIN {X 0,Y 375.493,Z 429.392,A -85,B 0,C 180,E1 -12310.041,E2 -12310.041} C_VEL
LIN {X 0,Y 378.065,Z 445.268,A -85,B 0,C 180,E1 -12310.727,E2 -12310.727} C_VEL
LIN {X 0,Y 379.395,Z 459.052,A -85,B 0,C 180,E1 -12311.526,E2 -12311.526} C_VEL
LIN {X 0,Y 379.697,Z 470.565,A -85,B 0,C 180,E1 -12312.357,E2 -12312.357} C_VEL
LIN {X 0,Y 379.622,Z 478.538,A -85,B 0,C 180,E1 -12313.048,E2 -12313.048} C_VEL
LIN {X 0,Y 378.286,Z 490.219,A -85,B 0,C 180,E1 -12314.235,E2 -12314.235} C_VEL
LIN {X 0,Y 377.225,Z 500.536,A -85,B 0,C 180,E1 -12315.556,E2 -12315.556} C_VEL
LIN {X 0,Y 376.539,Z 508.384,A -85,B 0,C 180,E1 -12316.784,E2 -12316.784} C_VEL
LIN {X 0,Y 375.706,Z 516.873,A -85,B 0,C 180,E1 -12318.4,E2 -12318.4} C_VEL
LIN {X 0,Y 375.176,Z 523.763,A -85,B 0,C 180,E1 -12320.022,E2 -12320.022} C_VEL
LIN {X 0,Y 374.94,Z 530.153,A -85,B 0,C 180,E1 -12321.919,E2 -12321.919} C_VEL
LIN {X 0,Y 374.932,Z 534.347,A -85,B 0,C 180,E1 -12323.543,E2 -12323.543} C_VEL
LIN {X 0,Y 374.972,Z 536.539,A -85,B 0,C 180,E1 -12324.623,E2 -12324.623} C_VEL
LIN {X 0,Y 375.098,Z 538.298,A -85,B 0,C 180,E1 -12325.703,E2 -12325.703} C_VEL
LIN {X 0,Y 375.23,Z 539.645,A -85,B 0,C 180,E1 -12326.78,E2 -12326.78} C_VEL
LIN {X 0,Y 375.157,Z 540.559,A -85,B 0,C 180,E1 -12327.854,E2 -12327.854} C_VEL
LIN {X 0,Y 375.182,Z 541.037,A -85,B 0,C 180,E1 -12328.927,E2 -12328.927} C_VEL
LIN {X 0,Y 375.243,Z 541.114,A -85,B 0,C 180,E1 -12330.001,E2 -12330.001} C_VEL
LIN {X 0,Y 375.211,Z 540.782,A -85,B 0,C 180,E1 -12331.074,E2 -12331.074} C_VEL
LIN {X 0,Y 375.201,Z 540.05,A -85,B 0,C 180,E1 -12332.148,E2 -12332.148} C_VEL
LIN {X 0,Y 375.254,Z 538.871,A -85,B 0,C 180,E1 -12333.222,E2 -12333.222} C_VEL
LIN {X 0,Y 375.115,Z 536.28,A -85,B 0,C 180,E1 -12334.837,E2 -12334.837} C_VEL
LIN {X 0,Y 375.023,Z 532.06,A -85,B 0,C 180,E1 -12336.67,E2 -12336.67} C_VEL
LIN {X 0,Y 375.041,Z 525.987,A -85,B 0,C 180,E1 -12338.623,E2 -12338.623} C_VEL
LIN {X 0,Y 375.228,Z 519.482,A -85,B 0,C 180,E1 -12340.25,E2 -12340.25} C_VEL
LIN {X 0,Y 375.777,Z 511.368,A -85,B 0,C 180,E1 -12341.873,E2 -12341.873} C_VEL
LIN {X 0,Y 376.523,Z 501.479,A -85,B 0,C 180,E1 -12343.465,E2 -12343.465} C_VEL
LIN {X 0,Y 377.227,Z 492.276,A -85,B 0,C 180,E1 -12344.664,E2 -12344.664} C_VEL
LIN {X 0,Y 378.084,Z 481.773,A -85,B 0,C 180,E1 -12345.776,E2 -12345.776} C_VEL
LIN {X 0,Y 378.613,Z 472.484,A -85,B 0,C 180,E1 -12346.583,E2 -12346.583} C_VEL
LIN {X 0,Y 377.969,Z 459.592,A -85,B 0,C 180,E1 -12347.499,E2 -12347.499} C_VEL
LIN {X 0,Y 376.938,Z 446.399,A -85,B 0,C 180,E1 -12348.211,E2 -12348.211} C_VEL
LIN {X 0,Y 375.543,Z 433.041,A -85,B 0,C 180,E1 -12348.71,E2 -12348.71} C_VEL
LIN {X 0,Y 375.266,Z 430.29,A -85,B 0,C 180,E1 -12348.813,E2 -12348.813} C_VEL
LIN {X 0,Y 375.73,Z 418.615,A -85,B 0,C 180,E1 -12352.548,E2 -12352.548} C_VEL
LIN {X 0,Y 376.327,Z 406.911,A -85,B 0,C 180,E1 -12356.31,E2 -12356.31} C_VEL
LIN {X 0,Y 377.056,Z 396.778,A -85,B 0,C 180,E1 -12359.601,E2 -12359.601} C_VEL
LIN {X 0,Y 377.972,Z 385.098,A -85,B 0,C 180,E1 -12363.49,E2 -12363.49} C_VEL
LIN {X 0,Y 378.797,Z 376.534,A -85,B 0,C 180,E1 -12366.422,E2 -12366.422} C_VEL
LIN {X 0,Y 378.6,Z 372.757,A -85,B 0,C 180,E1 -12367.777,E2 -12367.777} C_VEL
LIN {X 0,Y 377.227,Z 365.068,A -85,B 0,C 180,E1 -12370.699,E2 -12370.699} C_VEL
LIN {X 0,Y 376.006,Z 358.651,A -85,B 0,C 180,E1 -12373.316,E2 -12373.316} C_VEL
LIN {X 0,Y 375.938,Z 358.659,A -85,B 0,C 180,E1 -12376.811,E2 -12376.811} C_VEL
LIN {X 0,Y 375.967,Z 358.652,A -85,B 0,C 180,E1 -12380.538,E2 -12380.538} C_VEL
LIN {X 0,Y 375.968,Z 358.652,A -85,B 0,C 180,E1 -12383.496,E2 -12383.496} C_VEL
LIN {X 0,Y 375.964,Z 358.651,A -85,B 0,C 180,E1 -12385.889,E2 -12385.889} C_VEL
LIN {X 0,Y 375.969,Z 358.65,A -85,B 0,C 180,E1 -12389.688,E2 -12389.688} C_VEL
LIN {X 0,Y 376.025,Z 358.644,A -85,B 0,C 180,E1 -12393.348,E2 -12393.348} C_VEL
LIN {X 0,Y 376.002,Z 358.65,A -85,B 0,C 180,E1 -12396.889,E2 -12396.889} C_VEL
LIN {X 0,Y 376.003,Z 358.65,A -85,B 0,C 180,E1 -12400.34,E2 -12400.34} C_VEL
LIN {X 0,Y 376.034,Z 358.642,A -85,B 0,C 180,E1 -12403.719,E2 -12403.719} C_VEL
LIN {X 0,Y 376.109,Z 358.634,A -85,B 0,C 180,E1 -12407.042,E2 -12407.042} C_VEL
LIN {X 0,Y 376.124,Z 358.636,A -85,B 0,C 180,E1 -12410.319,E2 -12410.319} C_VEL
LIN {X 0,Y 376.237,Z 358.622,A -85,B 0,C 180,E1 -12412.487,E2 -12412.487} C_VEL
LIN {X 0,Y 376.177,Z 358.628,A -85,B 0,C 180,E1 -12414.64,E2 -12414.64} C_VEL
LIN {X 0,Y 376.357,Z 358.604,A -85,B 0,C 180,E1 -12417.86,E2 -12417.86} C_VEL
LIN {X 0,Y 376.495,Z 358.589,A -85,B 0,C 180,E1 -12420,E2 -12420} C_VEL
LIN {X 0,Y 376.19,Z 358.623,A -85,B 0,C 180,E1 -12423.213,E2 -12423.213} C_VEL
LIN {X 0,Y 376.239,Z 358.618,A -85,B 0,C 180,E1 -12426.641,E2 -12426.641} C_VEL
LIN {X 0,Y 376.211,Z 358.621,A -85,B 0,C 180,E1 -12428.595,E2 -12428.595} C_VEL
LIN {X 0,Y 376.057,Z 358.644,A -85,B 0,C 180,E1 -12431.863,E2 -12431.863} C_VEL
LIN {X 0,Y 376.065,Z 358.638,A -85,B 0,C 180,E1 -12435.167,E2 -12435.167} C_VEL
LIN {X 0,Y 376.03,Z 358.643,A -85,B 0,C 180,E1 -12438.526,E2 -12438.526} C_VEL
LIN {X 0,Y 375.969,Z 358.655,A -85,B 0,C 180,E1 -12441.954,E2 -12441.954} C_VEL
LIN {X 0,Y 376.013,Z 358.648,A -85,B 0,C 180,E1 -12445.461,E2 -12445.461} C_VEL
LIN {X 0,Y 375.967,Z 358.651,A -85,B 0,C 180,E1 -12449.08,E2 -12449.08} C_VEL
LIN {X 0,Y 375.955,Z 358.652,A -85,B 0,C 180,E1 -12452.828,E2 -12452.828} C_VEL
LIN {X 0,Y 375.964,Z 358.656,A -85,B 0,C 180,E1 -12455.415,E2 -12455.415} C_VEL
LIN {X 0,Y 375.98,Z 358.649,A -85,B 0,C 180,E1 -12458.27,E2 -12458.27} C_VEL
LIN {X 0,Y 375.941,Z 358.658,A -85,B 0,C 180,E1 -12461.601,E2 -12461.601} C_VEL
LIN {X 0,Y 375.959,Z 358.657,A -85,B 0,C 180,E1 -12465.264,E2 -12465.264} C_VEL
LIN {X 0,Y 375.946,Z 358.658,A -85,B 0,C 180,E1 -12469.133,E2 -12469.133} C_VEL
LIN {X 0,Y 375.97,Z 358.651,A -85,B 0,C 180,E1 -12471.911,E2 -12471.911} C_VEL
LIN {X 0,Y 375.986,Z 358.653,A -85,B 0,C 180,E1 -12475.332,E2 -12475.332} C_VEL
LIN {X 0,Y 375.964,Z 358.652,A -85,B 0,C 180,E1 -12478.438,E2 -12478.438} C_VEL
LIN {X 0,Y 375.989,Z 358.648,A -85,B 0,C 180,E1 -12482.14,E2 -12482.14} C_VEL
LIN {X 0,Y 376.013,Z 358.647,A -85,B 0,C 180,E1 -12484.539,E2 -12484.539} C_VEL
LIN {X 0,Y 375.97,Z 358.65,A -85,B 0,C 180,E1 -12488.045,E2 -12488.045} C_VEL
LIN {X 0,Y 376.015,Z 358.645,A -85,B 0,C 180,E1 -12491.473,E2 -12491.473} C_VEL
LIN {X 0,Y 376.065,Z 358.644,A -85,B 0,C 180,E1 -12494.832,E2 -12494.832} C_VEL
LIN {X 0,Y 376.057,Z 358.64,A -85,B 0,C 180,E1 -12498.136,E2 -12498.136} C_VEL
LIN {X 0,Y 376.122,Z 358.678,A -85,B 0,C 180,E1 -12499.921,E2 -12499.921} C_VEL
LIN {X 0,Y 379.822,Z 370.944,A -85,B 0,C 180,E1 -12500.763,E2 -12500.763} C_VEL
LIN {X 0,Y 381.189,Z 376.454,A -85,B 0,C 180,E1 -12501.203,E2 -12501.203} C_VEL
LIN {X 0,Y 380.565,Z 386.98,A -85,B 0,C 180,E1 -12502.038,E2 -12502.038} C_VEL
LIN {X 0,Y 379.831,Z 397.496,A -85,B 0,C 180,E1 -12503.092,E2 -12503.092} C_VEL
LIN {X 0,Y 379.038,Z 408.029,A -85,B 0,C 180,E1 -12504.413,E2 -12504.413} C_VEL
LIN {X 0,Y 378.33,Z 416.593,A -85,B 0,C 180,E1 -12505.738,E2 -12505.738} C_VEL
LIN {X 0,Y 377.522,Z 424.95,A -85,B 0,C 180,E1 -12507.332,E2 -12507.332} C_VEL
LIN {X 0,Y 376.866,Z 431.649,A -85,B 0,C 180,E1 -12508.931,E2 -12508.931} C_VEL
LIN {X 0,Y 376.419,Z 437.003,A -85,B 0,C 180,E1 -12510.534,E2 -12510.534} C_VEL
LIN {X 0,Y 376.056,Z 441.211,A -85,B 0,C 180,E1 -12512.141,E2 -12512.141} C_VEL
LIN {X 0,Y 375.777,Z 443.461,A -85,B 0,C 180,E1 -12513.216,E2 -12513.216} C_VEL
LIN {X 0,Y 375.696,Z 445.251,A -85,B 0,C 180,E1 -12514.29,E2 -12514.29} C_VEL
LIN {X 0,Y 375.694,Z 446.589,A -85,B 0,C 180,E1 -12515.366,E2 -12515.366} C_VEL
LIN {X 0,Y 375.651,Z 448.147,A -85,B 0,C 180,E1 -12517.524,E2 -12517.524} C_VEL
LIN {X 0,Y 375.648,Z 448.338,A -85,B 0,C 180,E1 -12518.607,E2 -12518.607} C_VEL
LIN {X 0,Y 375.741,Z 447.519,A -85,B 0,C 180,E1 -12520.78,E2 -12520.78} C_VEL
LIN {X 0,Y 375.898,Z 446.53,A -85,B 0,C 180,E1 -12521.867,E2 -12521.867} C_VEL
LIN {X 0,Y 376.382,Z 443.627,A -85,B 0,C 180,E1 -12523.837,E2 -12523.837} C_VEL
LIN {X 0,Y 376.923,Z 439.582,A -85,B 0,C 180,E1 -12525.685,E2 -12525.685} C_VEL
LIN {X 0,Y 377.534,Z 434.791,A -85,B 0,C 180,E1 -12527.328,E2 -12527.328} C_VEL
LIN {X 0,Y 378.315,Z 428.916,A -85,B 0,C 180,E1 -12528.915,E2 -12528.915} C_VEL
LIN {X 0,Y 379.118,Z 422.418,A -85,B 0,C 180,E1 -12530.339,E2 -12530.339} C_VEL
LIN {X 0,Y 380.182,Z 413.598,A -85,B 0,C 180,E1 -12531.904,E2 -12531.904} C_VEL
LIN {X 0,Y 381.152,Z 403.374,A -85,B 0,C 180,E1 -12533.355,E2 -12533.355} C_VEL
LIN {X 0,Y 382.093,Z 393.766,A -85,B 0,C 180,E1 -12534.446,E2 -12534.446} C_VEL
LIN {X 0,Y 383.042,Z 382.615,A -85,B 0,C 180,E1 -12535.461,E2 -12535.461} C_VEL
LIN {X 0,Y 383.228,Z 379.991,A -85,B 0,C 180,E1 -12535.662,E2 -12535.662} C_VEL
LIN {X 0,Y 380.397,Z 370.815,A -85,B 0,C 180,E1 -12536.512,E2 -12536.512} C_VEL
LIN {X 0,Y 378.017,Z 364.123,A -85,B 0,C 180,E1 -12537.069,E2 -12537.069} C_VEL
LIN {X 0,Y 376.87,Z 361.853,A -85,B 0,C 180,E1 -12537.363,E2 -12537.363} C_VEL
LIN {X 0,Y 375.164,Z 360.097,A -85,B 0,C 180,E1 -12537.878,E2 -12537.878} C_VEL
LIN {X 0,Y 372.897,Z 359.182,A -85,B 0,C 180,E1 -12538.692,E2 -12538.692} C_VEL
LIN {X 0,Y 369.853,Z 359.419,A -85,B 0,C 180,E1 -12540.257,E2 -12540.257} C_VEL
LIN {X 0,Y 368.953,Z 359.532,A -85,B 0,C 180,E1 -12541.25,E2 -12541.25} C_VEL
LIN {X 0,Y 368.883,Z 359.536,A -85,B 0,C 180,E1 -12541.584,E2 -12541.584} C_VEL
LIN {X 0,Y 368.929,Z 359.534,A -85,B 0,C 180,E1 -12545,E2 -12545} C_VEL
LIN {X 0,Y 368.909,Z 359.535,A -85,B 0,C 180,E1 -12548.639,E2 -12548.639} C_VEL
LIN {X 0,Y 368.881,Z 359.535,A -85,B 0,C 180,E1 -12552.009,E2 -12552.009} C_VEL
LIN {X 0,Y 368.881,Z 359.538,A -85,B 0,C 180,E1 -12555.175,E2 -12555.175} C_VEL
LIN {X 0,Y 368.909,Z 359.536,A -85,B 0,C 180,E1 -12558.181,E2 -12558.181} C_VEL
LIN {X 0,Y 368.912,Z 359.535,A -85,B 0,C 180,E1 -12561.358,E2 -12561.358} C_VEL
LIN {X 0,Y 368.935,Z 359.53,A -85,B 0,C 180,E1 -12565.146,E2 -12565.146} C_VEL
LIN {X 0,Y 368.926,Z 359.506,A -85,B 0,C 180,E1 -12569.046,E2 -12569.046} C_VEL
LIN {X 0,Y 368.984,Z 359.507,A -85,B 0,C 180,E1 -12571.564,E2 -12571.564} C_VEL
LIN {X 0,Y 368.955,Z 359.527,A -85,B 0,C 180,E1 -12575.224,E2 -12575.224} C_VEL
LIN {X 0,Y 368.934,Z 359.529,A -85,B 0,C 180,E1 -12578.973,E2 -12578.973} C_VEL
LIN {X 0,Y 368.987,Z 359.515,A -85,B 0,C 180,E1 -12582.257,E2 -12582.257} C_VEL
LIN {X 0,Y 369.034,Z 359.517,A -85,B 0,C 180,E1 -12586.227,E2 -12586.227} C_VEL
LIN {X 0,Y 369.069,Z 359.511,A -85,B 0,C 180,E1 -12590.131,E2 -12590.131} C_VEL
LIN {X 0,Y 369.185,Z 359.498,A -85,B 0,C 180,E1 -12592.342,E2 -12592.342} C_VEL
LIN {X 0,Y 369.142,Z 359.494,A -85,B 0,C 180,E1 -12594.537,E2 -12594.537} C_VEL
LIN {X 0,Y 369.316,Z 359.482,A -85,B 0,C 180,E1 -12597.819,E2 -12597.819} C_VEL
LIN {X 0,Y 369.457,Z 359.456,A -85,B 0,C 180,E1 -12600,E2 -12600} C_VEL
LIN {X 0,Y 369.316,Z 359.483,A -85,B 0,C 180,E1 -12602.181,E2 -12602.181} C_VEL
LIN {X 0,Y 369.205,Z 359.496,A -85,B 0,C 180,E1 -12606.558,E2 -12606.558} C_VEL
LIN {X 0,Y 369.133,Z 359.503,A -85,B 0,C 180,E1 -12608.761,E2 -12608.761} C_VEL
LIN {X 0,Y 369.002,Z 359.522,A -85,B 0,C 180,E1 -12612.093,E2 -12612.093} C_VEL
LIN {X 0,Y 368.994,Z 359.523,A -85,B 0,C 180,E1 -12615.465,E2 -12615.465} C_VEL
LIN {X 0,Y 368.978,Z 359.525,A -85,B 0,C 180,E1 -12618.893,E2 -12618.893} C_VEL
LIN {X 0,Y 368.928,Z 359.533,A -85,B 0,C 180,E1 -12622.395,E2 -12622.395} C_VEL
LIN {X 0,Y 368.996,Z 359.525,A -85,B 0,C 180,E1 -12625.98,E2 -12625.98} C_VEL
LIN {X 0,Y 368.964,Z 359.529,A -85,B 0,C 180,E1 -12628.814,E2 -12628.814} C_VEL
LIN {X 0,Y 368.896,Z 359.537,A -85,B 0,C 180,E1 -12632.238,E2 -12632.238} C_VEL
LIN {X 0,Y 368.926,Z 359.533,A -85,B 0,C 180,E1 -12635.002,E2 -12635.002} C_VEL
LIN {X 0,Y 368.91,Z 359.523,A -85,B 0,C 180,E1 -12638.642,E2 -12638.642} C_VEL
LIN {X 0,Y 368.939,Z 359.522,A -85,B 0,C 180,E1 -12642.02,E2 -12642.02} C_VEL
LIN {X 0,Y 368.984,Z 359.662,A -85,B 0,C 180,E1 -12643.85,E2 -12643.85} C_VEL
LIN {X 0,Y 370.325,Z 366.25,A -85,B 0,C 180,E1 -12646.906,E2 -12646.906} C_VEL
LIN {X 0,Y 371.703,Z 373.345,A -85,B 0,C 180,E1 -12649.996,E2 -12649.996} C_VEL
LIN {X 0,Y 372.683,Z 379.164,A -85,B 0,C 180,E1 -12652.376,E2 -12652.376} C_VEL
LIN {X 0,Y 372.566,Z 382.239,A -85,B 0,C 180,E1 -12653.545,E2 -12653.545} C_VEL
LIN {X 0,Y 371.276,Z 392.736,A -85,B 0,C 180,E1 -12657.352,E2 -12657.352} C_VEL
LIN {X 0,Y 370.164,Z 403.829,A -85,B 0,C 180,E1 -12661.242,E2 -12661.242} C_VEL
LIN {X 0,Y 369.344,Z 413.786,A -85,B 0,C 180,E1 -12664.651,E2 -12664.651} C_VEL
LIN {X 0,Y 368.658,Z 424.252,A -85,B 0,C 180,E1 -12668.178,E2 -12668.178} C_VEL
LIN {X 0,Y 368.45,Z 428.477,A -85,B 0,C 180,E1 -12669.591,E2 -12669.591} C_VEL
LIN {X 0,Y 371.024,Z 443.896,A -85,B 0,C 180,E1 -12670.269,E2 -12670.269} C_VEL
LIN {X 0,Y 372.289,Z 455.628,A -85,B 0,C 180,E1 -12670.946,E2 -12670.946} C_VEL
LIN {X 0,Y 372.831,Z 466.774,A -85,B 0,C 180,E1 -12671.737,E2 -12671.737} C_VEL
LIN {X 0,Y 372.816,Z 478.169,A -85,B 0,C 180,E1 -12672.729,E2 -12672.729} C_VEL
LIN {X 0,Y 371.432,Z 489.756,A -85,B 0,C 180,E1 -12673.936,E2 -12673.936} C_VEL
LIN {X 0,Y 370.355,Z 499.522,A -85,B 0,C 180,E1 -12675.213,E2 -12675.213} C_VEL
LIN {X 0,Y 369.615,Z 507.769,A -85,B 0,C 180,E1 -12676.531,E2 -12676.531} C_VEL
LIN {X 0,Y 368.827,Z 514.942,A -85,B 0,C 180,E1 -12677.902,E2 -12677.902} C_VEL
LIN {X 0,Y 368.171,Z 522.012,A -85,B 0,C 180,E1 -12679.553,E2 -12679.553} C_VEL
LIN {X 0,Y 367.908,Z 527.736,A -85,B 0,C 180,E1 -12681.21,E2 -12681.21} C_VEL
LIN {X 0,Y 367.819,Z 532.27,A -85,B 0,C 180,E1 -12682.866,E2 -12682.866} C_VEL
LIN {X 0,Y 367.908,Z 535.735,A -85,B 0,C 180,E1 -12684.52,E2 -12684.52} C_VEL
LIN {X 0,Y 368.023,Z 537.479,A -85,B 0,C 180,E1 -12685.62,E2 -12685.62} C_VEL
LIN {X 0,Y 368.164,Z 538.814,A -85,B 0,C 180,E1 -12686.718,E2 -12686.718} C_VEL
LIN {X 0,Y 368.108,Z 539.71,A -85,B 0,C 180,E1 -12687.812,E2 -12687.812} C_VEL
LIN {X 0,Y 368.131,Z 540.169,A -85,B 0,C 180,E1 -12688.907,E2 -12688.907} C_VEL
LIN {X 0,Y 368.197,Z 540.234,A -85,B 0,C 180,E1 -12690.001,E2 -12690.001} C_VEL
LIN {X 0,Y 368.163,Z 539.889,A -85,B 0,C 180,E1 -12691.095,E2 -12691.095} C_VEL
LIN {X 0,Y 368.153,Z 539.138,A -85,B 0,C 180,E1 -12692.189,E2 -12692.189} C_VEL
LIN {X 0,Y 368.21,Z 537.937,A -85,B 0,C 180,E1 -12693.283,E2 -12693.283} C_VEL
LIN {X 0,Y 368.044,Z 535.311,A -85,B 0,C 180,E1 -12694.93,E2 -12694.93} C_VEL
LIN {X 0,Y 367.964,Z 531.341,A -85,B 0,C 180,E1 -12696.693,E2 -12696.693} C_VEL
LIN {X 0,Y 367.951,Z 526.818,A -85,B 0,C 180,E1 -12698.237,E2 -12698.237} C_VEL
LIN {X 0,Y 368.144,Z 519.565,A -85,B 0,C 180,E1 -12700.172,E2 -12700.172} C_VEL
LIN {X 0,Y 368.661,Z 511.738,A -85,B 0,C 180,E1 -12701.826,E2 -12701.826} C_VEL
LIN {X 0,Y 369.407,Z 502.253,A -85,B 0,C 180,E1 -12703.425,E2 -12703.425} C_VEL
LIN {X 0,Y 370.139,Z 492.869,A -85,B 0,C 180,E1 -12704.713,E2 -12704.713} C_VEL
LIN {X 0,Y 371.081,Z 481.817,A -85,B 0,C 180,E1 -12705.94,E2 -12705.94} C_VEL
LIN {X 0,Y 371.649,Z 474.312,A -85,B 0,C 180,E1 -12706.621,E2 -12706.621} C_VEL
LIN {X 0,Y 371.121,Z 462.12,A -85,B 0,C 180,E1 -12707.567,E2 -12707.567} C_VEL
LIN {X 0,Y 370.156,Z 448.9,A -85,B 0,C 180,E1 -12708.35,E2 -12708.35} C_VEL
LIN {X 0,Y 368.88,Z 435.497,A -85,B 0,C 180,E1 -12708.917,E2 -12708.917} C_VEL
LIN {X 0,Y 368.189,Z 429.513,A -85,B 0,C 180,E1 -12709.117,E2 -12709.117} C_VEL
LIN {X 0,Y 368.616,Z 419.395,A -85,B 0,C 180,E1 -12712.416,E2 -12712.416} C_VEL
LIN {X 0,Y 369.209,Z 408.586,A -85,B 0,C 180,E1 -12715.965,E2 -12715.965} C_VEL
LIN {X 0,Y 369.999,Z 397.672,A -85,B 0,C 180,E1 -12719.596,E2 -12719.596} C_VEL
LIN {X 0,Y 370.932,Z 386.122,A -85,B 0,C 180,E1 -12723.523,E2 -12723.523} C_VEL
LIN {X 0,Y 371.825,Z 377.469,A -85,B 0,C 180,E1 -12726.542,E2 -12726.542} C_VEL
LIN {X 0,Y 371.545,Z 373.558,A -85,B 0,C 180,E1 -12727.985,E2 -12727.985} C_VEL
LIN {X 0,Y 370.036,Z 365.243,A -85,B 0,C 180,E1 -12731.222,E2 -12731.222} C_VEL
LIN {X 0,Y 368.937,Z 359.534,A -85,B 0,C 180,E1 -12733.625,E2 -12733.625} C_VEL
LIN {X 0,Y 368.89,Z 359.537,A -85,B 0,C 180,E1 -12736.696,E2 -12736.696} C_VEL
LIN {X 0,Y 368.916,Z 359.529,A -85,B 0,C 180,E1 -12739.644,E2 -12739.644} C_VEL
LIN {X 0,Y 368.906,Z 359.534,A -85,B 0,C 180,E1 -12743.145,E2 -12743.145} C_VEL
LIN {X 0,Y 368.901,Z 359.533,A -85,B 0,C 180,E1 -12746.462,E2 -12746.462} C_VEL
LIN {X 0,Y 368.934,Z 359.53,A -85,B 0,C 180,E1 -12749.047,E2 -12749.047} C_VEL
LIN {X 0,Y 368.968,Z 359.528,A -85,B 0,C 180,E1 -12752.797,E2 -12752.797} C_VEL
LIN {X 0,Y 368.95,Z 359.525,A -85,B 0,C 180,E1 -12756.113,E2 -12756.113} C_VEL
LIN {X 0,Y 368.941,Z 359.526,A -85,B 0,C 180,E1 -12759.947,E2 -12759.947} C_VEL
LIN {X 0,Y 368.981,Z 359.52,A -85,B 0,C 180,E1 -12763.399,E2 -12763.399} C_VEL
LIN {X 0,Y 369.063,Z 359.513,A -85,B 0,C 180,E1 -12766.791,E2 -12766.791} C_VEL
LIN {X 0,Y 369.073,Z 359.512,A -85,B 0,C 180,E1 -12770.132,E2 -12770.132} C_VEL
LIN {X 0,Y 369.195,Z 359.499,A -85,B 0,C 180,E1 -12772.343,E2 -12772.343} C_VEL
LIN {X 0,Y 369.15,Z 359.504,A -85,B 0,C 180,E1 -12774.538,E2 -12774.538} C_VEL
LIN {X 0,Y 369.322,Z 359.48,A -85,B 0,C 180,E1 -12777.819,E2 -12777.819} C_VEL
LIN {X 0,Y 369.465,Z 359.464,A -85,B 0,C 180,E1 -12780,E2 -12780} C_VEL
LIN {X 0,Y 369.322,Z 359.484,A -85,B 0,C 180,E1 -12782.181,E2 -12782.181} C_VEL
LIN {X 0,Y 369.209,Z 359.493,A -85,B 0,C 180,E1 -12786.629,E2 -12786.629} C_VEL
LIN {X 0,Y 369.144,Z 359.501,A -85,B 0,C 180,E1 -12788.761,E2 -12788.761} C_VEL
LIN {X 0,Y 369.012,Z 359.522,A -85,B 0,C 180,E1 -12792.093,E2 -12792.093} C_VEL
LIN {X 0,Y 369.004,Z 359.519,A -85,B 0,C 180,E1 -12795.465,E2 -12795.465} C_VEL
LIN {X 0,Y 368.989,Z 359.519,A -85,B 0,C 180,E1 -12798.893,E2 -12798.893} C_VEL
LIN {X 0,Y 368.939,Z 359.527,A -85,B 0,C 180,E1 -12802.395,E2 -12802.395} C_VEL
LIN {X 0,Y 369.006,Z 359.521,A -85,B 0,C 180,E1 -12805.98,E2 -12805.98} C_VEL
LIN {X 0,Y 368.921,Z 359.533,A -85,B 0,C 180,E1 -12809.69,E2 -12809.69} C_VEL
LIN {X 0,Y 368.903,Z 359.532,A -85,B 0,C 180,E1 -12813.043,E2 -12813.043} C_VEL
LIN {X 0,Y 368.923,Z 359.528,A -85,B 0,C 180,E1 -12816.197,E2 -12816.197} C_VEL
LIN {X 0,Y 368.909,Z 359.531,A -85,B 0,C 180,E1 -12818.953,E2 -12818.953} C_VEL
LIN {X 0,Y 368.887,Z 359.533,A -85,B 0,C 180,E1 -12822.009,E2 -12822.009} C_VEL
LIN {X 0,Y 368.932,Z 359.531,A -85,B 0,C 180,E1 -12825.183,E2 -12825.183} C_VEL
LIN {X 0,Y 368.889,Z 359.532,A -85,B 0,C 180,E1 -12828.177,E2 -12828.177} C_VEL
LIN {X 0,Y 368.915,Z 359.533,A -85,B 0,C 180,E1 -12831.359,E2 -12831.359} C_VEL
LIN {X 0,Y 368.942,Z 359.531,A -85,B 0,C 180,E1 -12835.146,E2 -12835.146} C_VEL
LIN {X 0,Y 368.935,Z 359.532,A -85,B 0,C 180,E1 -12839.046,E2 -12839.046} C_VEL
LIN {X 0,Y 368.982,Z 359.522,A -85,B 0,C 180,E1 -12841.563,E2 -12841.563} C_VEL
LIN {X 0,Y 369.006,Z 359.517,A -85,B 0,C 180,E1 -12844.019,E2 -12844.019} C_VEL
LIN {X 0,Y 368.939,Z 359.526,A -85,B 0,C 180,E1 -12847.604,E2 -12847.604} C_VEL
LIN {X 0,Y 368.964,Z 359.526,A -85,B 0,C 180,E1 -12851.105,E2 -12851.105} C_VEL
LIN {X 0,Y 369.004,Z 359.522,A -85,B 0,C 180,E1 -12854.535,E2 -12854.535} C_VEL
LIN {X 0,Y 369.012,Z 359.517,A -85,B 0,C 180,E1 -12857.906,E2 -12857.906} C_VEL
LIN {X 0,Y 369.06,Z 359.548,A -85,B 0,C 180,E1 -12859.615,E2 -12859.615} C_VEL
LIN {X 0,Y 372.91,Z 372.108,A -85,B 0,C 180,E1 -12860.502,E2 -12860.502} C_VEL
LIN {X 0,Y 374.359,Z 377.44,A -85,B 0,C 180,E1 -12860.946,E2 -12860.946} C_VEL
LIN {X 0,Y 373.63,Z 388.933,A -85,B 0,C 180,E1 -12861.889,E2 -12861.889} C_VEL
LIN {X 0,Y 372.746,Z 400.403,A -85,B 0,C 180,E1 -12863.096,E2 -12863.096} C_VEL
LIN {X 0,Y 372.067,Z 409.626,A -85,B 0,C 180,E1 -12864.308,E2 -12864.308} C_VEL
LIN {X 0,Y 371.339,Z 418.066,A -85,B 0,C 180,E1 -12865.658,E2 -12865.658} C_VEL
LIN {X 0,Y 370.502,Z 426.28,A -85,B 0,C 180,E1 -12867.281,E2 -12867.281} C_VEL
LIN {X 0,Y 369.848,Z 432.894,A -85,B 0,C 180,E1 -12868.91,E2 -12868.91} C_VEL
LIN {X 0,Y 369.389,Z 438.175,A -85,B 0,C 180,E1 -12870.544,E2 -12870.544} C_VEL
LIN {X 0,Y 369.012,Z 442.315,A -85,B 0,C 180,E1 -12872.182,E2 -12872.182} C_VEL
LIN {X 0,Y 368.726,Z 444.533,A -85,B 0,C 180,E1 -12873.277,E2 -12873.277} C_VEL
LIN {X 0,Y 368.656,Z 446.258,A -85,B 0,C 180,E1 -12874.373,E2 -12874.373} C_VEL
LIN {X 0,Y 368.647,Z 447.568,A -85,B 0,C 180,E1 -12875.469,E2 -12875.469} C_VEL
LIN {X 0,Y 368.616,Z 449.063,A -85,B 0,C 180,E1 -12877.669,E2 -12877.669} C_VEL
LIN {X 0,Y 368.655,Z 448.949,A -85,B 0,C 180,E1 -12879.879,E2 -12879.879} C_VEL
LIN {X 0,Y 368.911,Z 447.293,A -85,B 0,C 180,E1 -12882.096,E2 -12882.096} C_VEL
LIN {X 0,Y 369.402,Z 444.499,A -85,B 0,C 180,E1 -12883.998,E2 -12883.998} C_VEL
LIN {X 0,Y 370.027,Z 440.19,A -85,B 0,C 180,E1 -12885.985,E2 -12885.985} C_VEL
LIN {X 0,Y 370.686,Z 435.327,A -85,B 0,C 180,E1 -12887.658,E2 -12887.658} C_VEL
LIN {X 0,Y 371.521,Z 429.372,A -85,B 0,C 180,E1 -12889.274,E2 -12889.274} C_VEL
LIN {X 0,Y 372.376,Z 422.782,A -85,B 0,C 180,E1 -12890.724,E2 -12890.724} C_VEL
LIN {X 0,Y 373.5,Z 413.951,A -85,B 0,C 180,E1 -12892.292,E2 -12892.292} C_VEL
LIN {X 0,Y 374.443,Z 404.512,A -85,B 0,C 180,E1 -12893.652,E2 -12893.652} C_VEL
LIN {X 0,Y 375.536,Z 393.656,A -85,B 0,C 180,E1 -12894.902,E2 -12894.902} C_VEL
LIN {X 0,Y 376.499,Z 382.69,A -85,B 0,C 180,E1 -12895.891,E2 -12895.891} C_VEL
LIN {X 0,Y 375.979,Z 379.38,A -85,B 0,C 180,E1 -12896.201,E2 -12896.201} C_VEL
LIN {X 0,Y 371.843,Z 367.222,A -85,B 0,C 180,E1 -12897.318,E2 -12897.318} C_VEL
LIN {X 0,Y 368.999,Z 359.786,A -85,B 0,C 180,E1 -12897.91,E2 -12897.91} C_VEL
LIN {X 0,Y 368.939,Z 359.533,A -85,B 0,C 180,E1 -12897.979,E2 -12897.979} C_VEL
LIN {X 0,Y 368.883,Z 359.536,A -85,B 0,C 180,E1 -12901.584,E2 -12901.584} C_VEL
LIN {X 0,Y 368.214,Z 359.626,A -85,B 0,C 180,E1 -12902.496,E2 -12902.496} C_VEL
LIN {X 0,Y 365.357,Z 359.979,A -85,B 0,C 180,E1 -12903.977,E2 -12903.977} C_VEL
LIN {X 0,Y 362.946,Z 360.28,A -85,B 0,C 180,E1 -12905.176,E2 -12905.176} C_VEL
LIN {X 0,Y 361.92,Z 360.406,A -85,B 0,C 180,E1 -12906.103,E2 -12906.103} C_VEL
LIN {X 0,Y 361.842,Z 360.413,A -85,B 0,C 180,E1 -12906.417,E2 -12906.417} C_VEL
LIN {X 0,Y 361.855,Z 360.411,A -85,B 0,C 180,E1 -12909.86,E2 -12909.86} C_VEL
LIN {X 0,Y 361.836,Z 360.415,A -85,B 0,C 180,E1 -12912.828,E2 -12912.828} C_VEL
LIN {X 0,Y 361.826,Z 360.417,A -85,B 0,C 180,E1 -12915.944,E2 -12915.944} C_VEL
LIN {X 0,Y 361.872,Z 360.412,A -85,B 0,C 180,E1 -12919.237,E2 -12919.237} C_VEL
LIN {X 0,Y 361.872,Z 360.41,A -85,B 0,C 180,E1 -12922.982,E2 -12922.982} C_VEL
LIN {X 0,Y 361.862,Z 360.409,A -85,B 0,C 180,E1 -12926.629,E2 -12926.629} C_VEL
LIN {X 0,Y 361.874,Z 360.379,A -85,B 0,C 180,E1 -12929.672,E2 -12929.672} C_VEL
LIN {X 0,Y 361.952,Z 360.397,A -85,B 0,C 180,E1 -12933.474,E2 -12933.474} C_VEL
LIN {X 0,Y 361.887,Z 360.398,A -85,B 0,C 180,E1 -12937.144,E2 -12937.144} C_VEL
LIN {X 0,Y 361.918,Z 360.402,A -85,B 0,C 180,E1 -12940.724,E2 -12940.724} C_VEL
LIN {X 0,Y 361.943,Z 360.4,A -85,B 0,C 180,E1 -12944.226,E2 -12944.226} C_VEL
LIN {X 0,Y 361.997,Z 360.392,A -85,B 0,C 180,E1 -12946.527,E2 -12946.527} C_VEL
LIN {X 0,Y 362.033,Z 360.387,A -85,B 0,C 180,E1 -12949.938,E2 -12949.938} C_VEL
LIN {X 0,Y 362.148,Z 360.375,A -85,B 0,C 180,E1 -12952.192,E2 -12952.192} C_VEL
LIN {X 0,Y 362.116,Z 360.369,A -85,B 0,C 180,E1 -12954.431,E2 -12954.431} C_VEL
LIN {X 0,Y 362.28,Z 360.359,A -85,B 0,C 180,E1 -12957.776,E2 -12957.776} C_VEL
LIN {X 0,Y 362.426,Z 360.331,A -85,B 0,C 180,E1 -12960,E2 -12960} C_VEL
LIN {X 0,Y 362.28,Z 360.36,A -85,B 0,C 180,E1 -12962.223,E2 -12962.223} C_VEL
LIN {X 0,Y 362.168,Z 360.372,A -85,B 0,C 180,E1 -12966.686,E2 -12966.686} C_VEL
LIN {X 0,Y 362.07,Z 360.382,A -85,B 0,C 180,E1 -12968.933,E2 -12968.933} C_VEL
LIN {X 0,Y 361.956,Z 360.399,A -85,B 0,C 180,E1 -12972.332,E2 -12972.332} C_VEL
LIN {X 0,Y 361.958,Z 360.396,A -85,B 0,C 180,E1 -12974.62,E2 -12974.62} C_VEL
LIN {X 0,Y 361.955,Z 360.396,A -85,B 0,C 180,E1 -12978.099,E2 -12978.099} C_VEL
LIN {X 0,Y 361.888,Z 360.409,A -85,B 0,C 180,E1 -12981.653,E2 -12981.653} C_VEL
LIN {X 0,Y 361.924,Z 360.407,A -85,B 0,C 180,E1 -12985.29,E2 -12985.29} C_VEL
LIN {X 0,Y 361.919,Z 360.407,A -85,B 0,C 180,E1 -12987.778,E2 -12987.778} C_VEL
LIN {X 0,Y 361.843,Z 360.416,A -85,B 0,C 180,E1 -12991.286,E2 -12991.286} C_VEL
LIN {X 0,Y 361.851,Z 360.413,A -85,B 0,C 180,E1 -12994.281,E2 -12994.281} C_VEL
LIN {X 0,Y 361.869,Z 360.41,A -85,B 0,C 180,E1 -12997.225,E2 -12997.225} C_VEL
LIN {X 0,Y 361.902,Z 360.402,A -85,B 0,C 180,E1 -13000.769,E2 -13000.769} C_VEL
LIN {X 0,Y 361.919,Z 360.512,A -85,B 0,C 180,E1 -13003.328,E2 -13003.328} C_VEL
LIN {X 0,Y 363.273,Z 367.156,A -85,B 0,C 180,E1 -13006.509,E2 -13006.509} C_VEL
LIN {X 0,Y 364.713,Z 374.499,A -85,B 0,C 180,E1 -13009.778,E2 -13009.778} C_VEL
LIN {X 0,Y 365.66,Z 379.884,A -85,B 0,C 180,E1 -13012.046,E2 -13012.046} C_VEL
LIN {X 0,Y 365.627,Z 383.399,A -85,B 0,C 180,E1 -13013.426,E2 -13013.426} C_VEL
LIN {X 0,Y 364.139,Z 395.22,A -85,B 0,C 180,E1 -13017.791,E2 -13017.791} C_VEL
LIN {X 0,Y 362.855,Z 407.853,A -85,B 0,C 180,E1 -13022.301,E2 -13022.301} C_VEL
LIN {X 0,Y 361.904,Z 420.053,A -85,B 0,C 180,E1 -13026.541,E2 -13026.541} C_VEL
LIN {X 0,Y 361.436,Z 427.513,A -85,B 0,C 180,E1 -13029.105,E2 -13029.105} C_VEL
LIN {X 0,Y 364.105,Z 443.158,A -85,B 0,C 180,E1 -13029.828,E2 -13029.828} C_VEL
LIN {X 0,Y 365.496,Z 456.064,A -85,B 0,C 180,E1 -13030.608,E2 -13030.608} C_VEL
LIN {X 0,Y 366.001,Z 468.322,A -85,B 0,C 180,E1 -13031.529,E2 -13031.529} C_VEL
LIN {X 0,Y 365.855,Z 479.244,A -85,B 0,C 180,E1 -13032.534,E2 -13032.534} C_VEL
LIN {X 0,Y 364.435,Z 490.411,A -85,B 0,C 180,E1 -13033.763,E2 -13033.763} C_VEL
LIN {X 0,Y 363.284,Z 500.409,A -85,B 0,C 180,E1 -13035.148,E2 -13035.148} C_VEL
LIN {X 0,Y 362.464,Z 508.661,A -85,B 0,C 180,E1 -13036.546,E2 -13036.546} C_VEL
LIN {X 0,Y 361.585,Z 516.794,A -85,B 0,C 180,E1 -13038.225,E2 -13038.225} C_VEL
LIN {X 0,Y 361.025,Z 523.367,A -85,B 0,C 180,E1 -13039.91,E2 -13039.91} C_VEL
LIN {X 0,Y 360.794,Z 528.642,A -85,B 0,C 180,E1 -13041.6,E2 -13041.6} C_VEL
LIN {X 0,Y 360.776,Z 533.123,A -85,B 0,C 180,E1 -13043.46,E2 -13043.46} C_VEL
LIN {X 0,Y 360.935,Z 536.661,A -85,B 0,C 180,E1 -13045.534,E2 -13045.534} C_VEL
LIN {X 0,Y 361.084,Z 537.984,A -85,B 0,C 180,E1 -13046.653,E2 -13046.653} C_VEL
LIN {X 0,Y 361.06,Z 538.858,A -85,B 0,C 180,E1 -13047.77,E2 -13047.77} C_VEL
LIN {X 0,Y 361.081,Z 539.302,A -85,B 0,C 180,E1 -13048.886,E2 -13048.886} C_VEL
LIN {X 0,Y 361.151,Z 539.354,A -85,B 0,C 180,E1 -13050.001,E2 -13050.001} C_VEL
LIN {X 0,Y 361.115,Z 538.995,A -85,B 0,C 180,E1 -13051.116,E2 -13051.116} C_VEL
LIN {X 0,Y 361.106,Z 538.221,A -85,B 0,C 180,E1 -13052.232,E2 -13052.232} C_VEL
LIN {X 0,Y 361.166,Z 537.001,A -85,B 0,C 180,E1 -13053.347,E2 -13053.347} C_VEL
LIN {X 0,Y 360.978,Z 534.34,A -85,B 0,C 180,E1 -13055.027,E2 -13055.027} C_VEL
LIN {X 0,Y 360.901,Z 530.634,A -85,B 0,C 180,E1 -13056.711,E2 -13056.711} C_VEL
LIN {X 0,Y 360.884,Z 525.774,A -85,B 0,C 180,E1 -13058.399,E2 -13058.399} C_VEL
LIN {X 0,Y 361.09,Z 518.479,A -85,B 0,C 180,E1 -13060.373,E2 -13060.373} C_VEL
LIN {X 0,Y 361.65,Z 510.591,A -85,B 0,C 180,E1 -13062.059,E2 -13062.059} C_VEL
LIN {X 0,Y 362.393,Z 501.293,A -85,B 0,C 180,E1 -13063.651,E2 -13063.651} C_VEL
LIN {X 0,Y 363.126,Z 492.687,A -85,B 0,C 180,E1 -13064.86,E2 -13064.86} C_VEL
LIN {X 0,Y 364.081,Z 481.79,A -85,B 0,C 180,E1 -13066.111,E2 -13066.111} C_VEL
LIN {X 0,Y 364.629,Z 474.443,A -85,B 0,C 180,E1 -13066.806,E2 -13066.806} C_VEL
LIN {X 0,Y 364.104,Z 461.472,A -85,B 0,C 180,E1 -13067.845,E2 -13067.845} C_VEL
LIN {X 0,Y 363.149,Z 448.209,A -85,B 0,C 180,E1 -13068.651,E2 -13068.651} C_VEL
LIN {X 0,Y 361.814,Z 434.298,A -85,B 0,C 180,E1 -13069.253,E2 -13069.253} C_VEL
LIN {X 0,Y 361.144,Z 428.663,A -85,B 0,C 180,E1 -13069.431,E2 -13069.431} C_VEL
LIN {X 0,Y 361.583,Z 418.378,A -85,B 0,C 180,E1 -13072.877,E2 -13072.877} C_VEL
LIN {X 0,Y 362.212,Z 407.599,A -85,B 0,C 180,E1 -13076.505,E2 -13076.505} C_VEL
LIN {X 0,Y 362.959,Z 398.105,A -85,B 0,C 180,E1 -13079.735,E2 -13079.735} C_VEL
LIN {X 0,Y 363.839,Z 387.813,A -85,B 0,C 180,E1 -13083.313,E2 -13083.313} C_VEL
LIN {X 0,Y 364.823,Z 378.395,A -85,B 0,C 180,E1 -13086.67,E2 -13086.67} C_VEL
LIN {X 0,Y 364.538,Z 374.622,A -85,B 0,C 180,E1 -13088.094,E2 -13088.094} C_VEL
LIN {X 0,Y 363.162,Z 366.945,A -85,B 0,C 180,E1 -13091.147,E2 -13091.147} C_VEL
LIN {X 0,Y 361.873,Z 360.413,A -85,B 0,C 180,E1 -13093.962,E2 -13093.962} C_VEL
LIN {X 0,Y 361.84,Z 360.411,A -85,B 0,C 180,E1 -13097.569,E2 -13097.569} C_VEL
LIN {X 0,Y 361.874,Z 360.411,A -85,B 0,C 180,E1 -13100.974,E2 -13100.974} C_VEL
LIN {X 0,Y 361.878,Z 360.409,A -85,B 0,C 180,E1 -13104.656,E2 -13104.656} C_VEL
LIN {X 0,Y 361.842,Z 360.411,A -85,B 0,C 180,E1 -13108.371,E2 -13108.371} C_VEL
LIN {X 0,Y 361.913,Z 360.402,A -85,B 0,C 180,E1 -13112.221,E2 -13112.221} C_VEL
LIN {X 0,Y 361.933,Z 360.404,A -85,B 0,C 180,E1 -13114.71,E2 -13114.71} C_VEL
LIN {X 0,Y 361.897,Z 360.406,A -85,B 0,C 180,E1 -13118.348,E2 -13118.348} C_VEL
LIN {X 0,Y 361.972,Z 360.395,A -85,B 0,C 180,E1 -13122.062,E2 -13122.062} C_VEL
LIN {X 0,Y 362.003,Z 360.392,A -85,B 0,C 180,E1 -13126.102,E2 -13126.102} C_VEL
LIN {X 0,Y 362.037,Z 360.387,A -85,B 0,C 180,E1 -13129.938,E2 -13129.938} C_VEL
LIN {X 0,Y 362.152,Z 360.375,A -85,B 0,C 180,E1 -13132.193,E2 -13132.193} C_VEL
LIN {X 0,Y 362.123,Z 360.38,A -85,B 0,C 180,E1 -13134.432,E2 -13134.432} C_VEL
LIN {X 0,Y 362.286,Z 360.356,A -85,B 0,C 180,E1 -13137.777,E2 -13137.777} C_VEL
LIN {X 0,Y 362.434,Z 360.34,A -85,B 0,C 180,E1 -13140,E2 -13140} C_VEL
LIN {X 0,Y 362.286,Z 360.36,A -85,B 0,C 180,E1 -13142.224,E2 -13142.224} C_VEL
LIN {X 0,Y 362.178,Z 360.369,A -85,B 0,C 180,E1 -13146.686,E2 -13146.686} C_VEL
LIN {X 0,Y 362.08,Z 360.38,A -85,B 0,C 180,E1 -13148.933,E2 -13148.933} C_VEL
LIN {X 0,Y 361.967,Z 360.397,A -85,B 0,C 180,E1 -13152.332,E2 -13152.332} C_VEL
LIN {X 0,Y 361.968,Z 360.394,A -85,B 0,C 180,E1 -13154.62,E2 -13154.62} C_VEL
LIN {X 0,Y 361.966,Z 360.398,A -85,B 0,C 180,E1 -13158.099,E2 -13158.099} C_VEL
LIN {X 0,Y 361.898,Z 360.407,A -85,B 0,C 180,E1 -13161.653,E2 -13161.653} C_VEL
LIN {X 0,Y 361.935,Z 360.4,A -85,B 0,C 180,E1 -13165.29,E2 -13165.29} C_VEL
LIN {X 0,Y 361.914,Z 360.406,A -85,B 0,C 180,E1 -13167.779,E2 -13167.779} C_VEL
LIN {X 0,Y 361.844,Z 360.415,A -85,B 0,C 180,E1 -13171.629,E2 -13171.629} C_VEL
LIN {X 0,Y 361.88,Z 360.409,A -85,B 0,C 180,E1 -13175.345,E2 -13175.345} C_VEL
LIN {X 0,Y 361.876,Z 360.407,A -85,B 0,C 180,E1 -13179.027,E2 -13179.027} C_VEL
LIN {X 0,Y 361.842,Z 360.411,A -85,B 0,C 180,E1 -13182.829,E2 -13182.829} C_VEL
LIN {X 0,Y 361.841,Z 360.411,A -85,B 0,C 180,E1 -13185.944,E2 -13185.944} C_VEL
LIN {X 0,Y 361.842,Z 360.415,A -85,B 0,C 180,E1 -13189.244,E2 -13189.244} C_VEL
LIN {X 0,Y 361.869,Z 360.408,A -85,B 0,C 180,E1 -13192.777,E2 -13192.777} C_VEL
LIN {X 0,Y 361.86,Z 360.408,A -85,B 0,C 180,E1 -13195.719,E2 -13195.719} C_VEL
LIN {X 0,Y 361.881,Z 360.406,A -85,B 0,C 180,E1 -13199.672,E2 -13199.672} C_VEL
LIN {X 0,Y 361.96,Z 360.397,A -85,B 0,C 180,E1 -13203.475,E2 -13203.475} C_VEL
LIN {X 0,Y 361.897,Z 360.407,A -85,B 0,C 180,E1 -13207.144,E2 -13207.144} C_VEL
LIN {X 0,Y 361.913,Z 360.406,A -85,B 0,C 180,E1 -13210.723,E2 -13210.723} C_VEL
LIN {X 0,Y 361.939,Z 360.401,A -85,B 0,C 180,E1 -13213.065,E2 -13213.065} C_VEL
LIN {X 0,Y 362.005,Z 360.393,A -85,B 0,C 180,E1 -13216.527,E2 -13216.527} C_VEL
LIN {X 0,Y 362.022,Z 360.452,A -85,B 0,C 180,E1 -13219.301,E2 -13219.301} C_VEL
LIN {X 0,Y 365.713,Z 372.341,A -85,B 0,C 180,E1 -13220.159,E2 -13220.159} C_VEL
LIN {X 0,Y 367.495,Z 379.007,A -85,B 0,C 180,E1 -13220.722,E2 -13220.722} C_VEL
LIN {X 0,Y 366.695,Z 390.859,A -85,B 0,C 180,E1 -13221.735,E2 -13221.735} C_VEL
LIN {X 0,Y 365.814,Z 402.135,A -85,B 0,C 180,E1 -13222.964,E2 -13222.964} C_VEL
LIN {X 0,Y 365.111,Z 411.206,A -85,B 0,C 180,E1 -13224.199,E2 -13224.199} C_VEL
LIN {X 0,Y 364.348,Z 419.498,A -85,B 0,C 180,E1 -13225.574,E2 -13225.574} C_VEL
LIN {X 0,Y 363.499,Z 427.604,A -85,B 0,C 180,E1 -13227.229,E2 -13227.229} C_VEL
LIN {X 0,Y 362.829,Z 434.136,A -85,B 0,C 180,E1 -13228.889,E2 -13228.889} C_VEL
LIN {X 0,Y 362.359,Z 439.343,A -85,B 0,C 180,E1 -13230.555,E2 -13230.555} C_VEL
LIN {X 0,Y 361.943,Z 443.421,A -85,B 0,C 180,E1 -13232.225,E2 -13232.225} C_VEL
LIN {X 0,Y 361.675,Z 445.59,A -85,B 0,C 180,E1 -13233.341,E2 -13233.341} C_VEL
LIN {X 0,Y 361.602,Z 448.546,A -85,B 0,C 180,E1 -13235.576,E2 -13235.576} C_VEL
LIN {X 0,Y 361.578,Z 449.874,A -85,B 0,C 180,E1 -13237.564,E2 -13237.564} C_VEL
LIN {X 0,Y 361.571,Z 450.062,A -85,B 0,C 180,E1 -13238.945,E2 -13238.945} C_VEL
LIN {X 0,Y 361.745,Z 449.122,A -85,B 0,C 180,E1 -13241.202,E2 -13241.202} C_VEL
LIN {X 0,Y 361.927,Z 448.039,A -85,B 0,C 180,E1 -13242.333,E2 -13242.333} C_VEL
LIN {X 0,Y 362.444,Z 445.348,A -85,B 0,C 180,E1 -13244.178,E2 -13244.178} C_VEL
LIN {X 0,Y 363.149,Z 440.802,A -85,B 0,C 180,E1 -13246.296,E2 -13246.296} C_VEL
LIN {X 0,Y 363.847,Z 435.867,A -85,B 0,C 180,E1 -13248.001,E2 -13248.001} C_VEL
LIN {X 0,Y 364.771,Z 429.594,A -85,B 0,C 180,E1 -13249.704,E2 -13249.704} C_VEL
LIN {X 0,Y 365.904,Z 421.662,A -85,B 0,C 180,E1 -13251.403,E2 -13251.403} C_VEL
LIN {X 0,Y 367.1,Z 412.055,A -85,B 0,C 180,E1 -13253.053,E2 -13253.053} C_VEL
LIN {X 0,Y 368.116,Z 402.334,A -85,B 0,C 180,E1 -13254.384,E2 -13254.384} C_VEL
LIN {X 0,Y 369.282,Z 390.601,A -85,B 0,C 180,E1 -13255.655,E2 -13255.655} C_VEL
LIN {X 0,Y 369.848,Z 382.975,A -85,B 0,C 180,E1 -13256.329,E2 -13256.329} C_VEL
LIN {X 0,Y 365.866,Z 370.813,A -85,B 0,C 180,E1 -13257.527,E2 -13257.527} C_VEL
LIN {X 0,Y 361.987,Z 360.836,A -85,B 0,C 180,E1 -13258.369,E2 -13258.369} C_VEL
LIN {X 0,Y 361.939,Z 360.402,A -85,B 0,C 180,E1 -13258.444,E2 -13258.444} C_VEL
LIN {X 0,Y 361.838,Z 360.416,A -85,B 0,C 180,E1 -13261.628,E2 -13261.628} C_VEL
LIN {X 0,Y 361.874,Z 360.414,A -85,B 0,C 180,E1 -13265.344,E2 -13265.344} C_VEL
LIN {X 0,Y 361.842,Z 360.413,A -85,B 0,C 180,E1 -13266.417,E2 -13266.417} C_VEL
LIN {X 0,Y 361.191,Z 360.498,A -85,B 0,C 180,E1 -13267.346,E2 -13267.346} C_VEL
LIN {X 0,Y 358.35,Z 360.855,A -85,B 0,C 180,E1 -13268.858,E2 -13268.858} C_VEL
LIN {X 0,Y 355.926,Z 361.156,A -85,B 0,C 180,E1 -13270.08,E2 -13270.08} C_VEL
LIN {X 0,Y 354.872,Z 361.284,A -85,B 0,C 180,E1 -13271.026,E2 -13271.026} C_VEL
LIN {X 0,Y 354.779,Z 361.293,A -85,B 0,C 180,E1 -13271.346,E2 -13271.346} C_VEL
LIN {X 0,Y 354.764,Z 361.294,A -85,B 0,C 180,E1 -13274.506,E2 -13274.506} C_VEL
LIN {X 0,Y 354.812,Z 361.29,A -85,B 0,C 180,E1 -13277.665,E2 -13277.665} C_VEL
LIN {X 0,Y 354.836,Z 361.286,A -85,B 0,C 180,E1 -13280.668,E2 -13280.668} C_VEL
LIN {X 0,Y 354.821,Z 361.285,A -85,B 0,C 180,E1 -13284.3,E2 -13284.3} C_VEL
LIN {X 0,Y 354.797,Z 361.283,A -85,B 0,C 180,E1 -13287.667,E2 -13287.667} C_VEL
LIN {X 0,Y 354.866,Z 361.253,A -85,B 0,C 180,E1 -13290.62,E2 -13290.62} C_VEL
LIN {X 0,Y 354.897,Z 361.277,A -85,B 0,C 180,E1 -13294.172,E2 -13294.172} C_VEL
LIN {X 0,Y 354.832,Z 361.282,A -85,B 0,C 180,E1 -13297.893,E2 -13297.893} C_VEL
LIN {X 0,Y 354.919,Z 361.267,A -85,B 0,C 180,E1 -13301.891,E2 -13301.891} C_VEL
LIN {X 0,Y 354.94,Z 361.273,A -85,B 0,C 180,E1 -13305.98,E2 -13305.98} C_VEL
LIN {X 0,Y 354.98,Z 361.265,A -85,B 0,C 180,E1 -13309.736,E2 -13309.736} C_VEL
LIN {X 0,Y 355.111,Z 361.252,A -85,B 0,C 180,E1 -13312.036,E2 -13312.036} C_VEL
LIN {X 0,Y 355.09,Z 361.244,A -85,B 0,C 180,E1 -13314.32,E2 -13314.32} C_VEL
LIN {X 0,Y 355.243,Z 361.235,A -85,B 0,C 180,E1 -13317.732,E2 -13317.732} C_VEL
LIN {X 0,Y 355.396,Z 361.207,A -85,B 0,C 180,E1 -13320,E2 -13320} C_VEL
LIN {X 0,Y 355.243,Z 361.236,A -85,B 0,C 180,E1 -13322.267,E2 -13322.267} C_VEL
LIN {X 0,Y 355.134,Z 361.248,A -85,B 0,C 180,E1 -13326.819,E2 -13326.819} C_VEL
LIN {X 0,Y 355.011,Z 361.259,A -85,B 0,C 180,E1 -13329.112,E2 -13329.112} C_VEL
LIN {X 0,Y 354.917,Z 361.275,A -85,B 0,C 180,E1 -13332.581,E2 -13332.581} C_VEL
LIN {X 0,Y 354.885,Z 361.281,A -85,B 0,C 180,E1 -13336.096,E2 -13336.096} C_VEL
LIN {X 0,Y 354.902,Z 361.277,A -85,B 0,C 180,E1 -13338.472,E2 -13338.472} C_VEL
LIN {X 0,Y 354.83,Z 361.289,A -85,B 0,C 180,E1 -13342.106,E2 -13342.106} C_VEL
LIN {X 0,Y 354.895,Z 361.281,A -85,B 0,C 180,E1 -13345.828,E2 -13345.828} C_VEL
LIN {X 0,Y 354.85,Z 361.287,A -85,B 0,C 180,E1 -13349.679,E2 -13349.679} C_VEL
LIN {X 0,Y 354.802,Z 361.292,A -85,B 0,C 180,E1 -13353.702,E2 -13353.702} C_VEL
LIN {X 0,Y 354.799,Z 361.292,A -85,B 0,C 180,E1 -13356.459,E2 -13356.459} C_VEL
LIN {X 0,Y 354.82,Z 361.282,A -85,B 0,C 180,E1 -13359.424,E2 -13359.424} C_VEL
LIN {X 0,Y 354.848,Z 361.353,A -85,B 0,C 180,E1 -13362.786,E2 -13362.786} C_VEL
LIN {X 0,Y 356.343,Z 368.598,A -85,B 0,C 180,E1 -13366.348,E2 -13366.348} C_VEL
LIN {X 0,Y 357.895,Z 376.595,A -85,B 0,C 180,E1 -13369.982,E2 -13369.982} C_VEL
LIN {X 0,Y 358.807,Z 382.795,A -85,B 0,C 180,E1 -13372.614,E2 -13372.614} C_VEL
LIN {X 0,Y 357.786,Z 390.564,A -85,B 0,C 180,E1 -13375.589,E2 -13375.589} C_VEL
LIN {X 0,Y 356.839,Z 398.465,A -85,B 0,C 180,E1 -13378.54,E2 -13378.54} C_VEL
LIN {X 0,Y 355.677,Z 410.114,A -85,B 0,C 180,E1 -13382.77,E2 -13382.77} C_VEL
LIN {X 0,Y 354.802,Z 421.069,A -85,B 0,C 180,E1 -13386.662,E2 -13386.662} C_VEL
LIN {X 0,Y 354.446,Z 426.816,A -85,B 0,C 180,E1 -13388.636,E2 -13388.636} C_VEL
LIN {X 0,Y 357.006,Z 441.155,A -85,B 0,C 180,E1 -13389.299,E2 -13389.299} C_VEL
LIN {X 0,Y 358.552,Z 453.93,A -85,B 0,C 180,E1 -13390.077,E2 -13390.077} C_VEL
LIN {X 0,Y 359.157,Z 466.335,A -85,B 0,C 180,E1 -13391.016,E2 -13391.016} C_VEL
LIN {X 0,Y 359.058,Z 478.9,A -85,B 0,C 180,E1 -13392.192,E2 -13392.192} C_VEL
LIN {X 0,Y 357.621,Z 489.932,A -85,B 0,C 180,E1 -13393.445,E2 -13393.445} C_VEL
LIN {X 0,Y 356.353,Z 499.854,A -85,B 0,C 180,E1 -13394.853,E2 -13394.853} C_VEL
LIN {X 0,Y 355.548,Z 508.052,A -85,B 0,C 180,E1 -13396.28,E2 -13396.28} C_VEL
LIN {X 0,Y 354.699,Z 514.875,A -85,B 0,C 180,E1 -13397.703,E2 -13397.703} C_VEL
LIN {X 0,Y 354.027,Z 521.638,A -85,B 0,C 180,E1 -13399.42,E2 -13399.42} C_VEL
LIN {X 0,Y 353.71,Z 527.883,A -85,B 0,C 180,E1 -13401.431,E2 -13401.431} C_VEL
LIN {X 0,Y 353.71,Z 532.572,A -85,B 0,C 180,E1 -13403.449,E2 -13403.449} C_VEL
LIN {X 0,Y 353.849,Z 535.844,A -85,B 0,C 180,E1 -13405.444,E2 -13405.444} C_VEL
LIN {X 0,Y 354.007,Z 537.155,A -85,B 0,C 180,E1 -13406.586,E2 -13406.586} C_VEL
LIN {X 0,Y 354.012,Z 538.005,A -85,B 0,C 180,E1 -13407.725,E2 -13407.725} C_VEL
LIN {X 0,Y 354.105,Z 538.475,A -85,B 0,C 180,E1 -13410.001,E2 -13410.001} C_VEL
LIN {X 0,Y 354.067,Z 538.101,A -85,B 0,C 180,E1 -13411.138,E2 -13411.138} C_VEL
LIN {X 0,Y 354.059,Z 537.299,A -85,B 0,C 180,E1 -13412.276,E2 -13412.276} C_VEL
LIN {X 0,Y 354.122,Z 536.063,A -85,B 0,C 180,E1 -13413.414,E2 -13413.414} C_VEL
LIN {X 0,Y 353.917,Z 533.368,A -85,B 0,C 180,E1 -13415.128,E2 -13415.128} C_VEL
LIN {X 0,Y 353.834,Z 529.626,A -85,B 0,C 180,E1 -13416.845,E2 -13416.845} C_VEL
LIN {X 0,Y 353.807,Z 524.725,A -85,B 0,C 180,E1 -13418.569,E2 -13418.569} C_VEL
LIN {X 0,Y 354.062,Z 517.391,A -85,B 0,C 180,E1 -13420.581,E2 -13420.581} C_VEL
LIN {X 0,Y 354.622,Z 509.426,A -85,B 0,C 180,E1 -13422.302,E2 -13422.302} C_VEL
LIN {X 0,Y 355.321,Z 501.303,A -85,B 0,C 180,E1 -13423.731,E2 -13423.731} C_VEL
LIN {X 0,Y 355.979,Z 493.578,A -85,B 0,C 180,E1 -13424.873,E2 -13424.873} C_VEL
LIN {X 0,Y 356.942,Z 483.043,A -85,B 0,C 180,E1 -13426.148,E2 -13426.148} C_VEL
LIN {X 0,Y 357.606,Z 474.56,A -85,B 0,C 180,E1 -13426.999,E2 -13426.999} C_VEL
LIN {X 0,Y 357.13,Z 461.841,A -85,B 0,C 180,E1 -13428.057,E2 -13428.057} C_VEL
LIN {X 0,Y 356.235,Z 448.551,A -85,B 0,C 180,E1 -13428.91,E2 -13428.91} C_VEL
LIN {X 0,Y 354.948,Z 434.938,A -85,B 0,C 180,E1 -13429.533,E2 -13429.533} C_VEL
LIN {X 0,Y 354.064,Z 427.731,A -85,B 0,C 180,E1 -13429.797,E2 -13429.797} C_VEL
LIN {X 0,Y 354.585,Z 417.354,A -85,B 0,C 180,E1 -13433.355,E2 -13433.355} C_VEL
LIN {X 0,Y 355.295,Z 406.481,A -85,B 0,C 180,E1 -13437.11,E2 -13437.11} C_VEL
LIN {X 0,Y 356.182,Z 395.739,A -85,B 0,C 180,E1 -13440.866,E2 -13440.866} C_VEL
LIN {X 0,Y 357.173,Z 384.785,A -85,B 0,C 180,E1 -13444.795,E2 -13444.795} C_VEL
LIN {X 0,Y 357.839,Z 379.133,A -85,B 0,C 180,E1 -13446.854,E2 -13446.854} C_VEL
LIN {X 0,Y 357.17,Z 373.609,A -85,B 0,C 180,E1 -13449.026,E2 -13449.026} C_VEL
LIN {X 0,Y 355.76,Z 365.962,A -85,B 0,C 180,E1 -13452.197,E2 -13452.197} C_VEL
LIN {X 0,Y 354.83,Z 361.291,A -85,B 0,C 180,E1 -13454.256,E2 -13454.256} C_VEL
LIN {X 0,Y 354.798,Z 361.288,A -85,B 0,C 180,E1 -13457.663,E2 -13457.663} C_VEL
LIN {X 0,Y 354.819,Z 361.287,A -85,B 0,C 180,E1 -13460.667,E2 -13460.667} C_VEL
LIN {X 0,Y 354.826,Z 361.284,A -85,B 0,C 180,E1 -13464.301,E2 -13464.301} C_VEL
LIN {X 0,Y 354.791,Z 361.288,A -85,B 0,C 180,E1 -13467.667,E2 -13467.667} C_VEL
LIN {X 0,Y 354.851,Z 361.28,A -85,B 0,C 180,E1 -13471.619,E2 -13471.619} C_VEL
LIN {X 0,Y 354.904,Z 361.275,A -85,B 0,C 180,E1 -13474.173,E2 -13474.173} C_VEL
LIN {X 0,Y 354.84,Z 361.282,A -85,B 0,C 180,E1 -13477.894,E2 -13477.894} C_VEL
LIN {X 0,Y 354.927,Z 361.271,A -85,B 0,C 180,E1 -13481.892,E2 -13481.892} C_VEL
LIN {X 0,Y 354.948,Z 361.27,A -85,B 0,C 180,E1 -13485.982,E2 -13485.982} C_VEL
LIN {X 0,Y 354.983,Z 361.264,A -85,B 0,C 180,E1 -13489.736,E2 -13489.736} C_VEL
LIN {X 0,Y 355.134,Z 361.248,A -85,B 0,C 180,E1 -13492.038,E2 -13492.038} C_VEL
LIN {X 0,Y 355.098,Z 361.255,A -85,B 0,C 180,E1 -13494.321,E2 -13494.321} C_VEL
LIN {X 0,Y 355.249,Z 361.232,A -85,B 0,C 180,E1 -13497.733,E2 -13497.733} C_VEL
LIN {X 0,Y 355.404,Z 361.215,A -85,B 0,C 180,E1 -13500,E2 -13500} C_VEL
LIN {X 0,Y 355.249,Z 361.236,A -85,B 0,C 180,E1 -13502.268,E2 -13502.268} C_VEL
LIN {X 0,Y 355.144,Z 361.244,A -85,B 0,C 180,E1 -13506.819,E2 -13506.819} C_VEL
